LIN {X 0,Y 411.188,Z 252.265,A -85,B 0,C 180,E1 -10477.975,E2 -10477.975} C_VEL
LIN {X 0,Y 411.151,Z 252.273,A -85,B 0,C 180,E1 -10481.226,E2 -10481.226} C_VEL
LIN {X 0,Y 411.176,Z 252.271,A -85,B 0,C 180,E1 -10484.491,E2 -10484.491} C_VEL
LIN {X 0,Y 411.189,Z 252.269,A -85,B 0,C 180,E1 -10488.196,E2 -10488.196} C_VEL
LIN {X 0,Y 411.23,Z 252.345,A -85,B 0,C 180,E1 -10489.137,E2 -10489.137} C_VEL
LIN {X 0,Y 412.077,Z 257.26,A -85,B 0,C 180,E1 -10492.122,E2 -10492.122} C_VEL
LIN {X 0,Y 412.498,Z 261.588,A -85,B 0,C 180,E1 -10494.6,E2 -10494.6} C_VEL
LIN {X 0,Y 412.052,Z 268.088,A -85,B 0,C 180,E1 -10498.079,E2 -10498.079} C_VEL
LIN {X 0,Y 411.534,Z 274.615,A -85,B 0,C 180,E1 -10501.434,E2 -10501.434} C_VEL
LIN {X 0,Y 411.14,Z 281.666,A -85,B 0,C 180,E1 -10504.956,E2 -10504.956} C_VEL
LIN {X 0,Y 410.788,Z 288.71,A -85,B 0,C 180,E1 -10508.418,E2 -10508.418} C_VEL
LIN {X 0,Y 410.454,Z 296.177,A -85,B 0,C 180,E1 -10512.049,E2 -10512.049} C_VEL
LIN {X 0,Y 410.432,Z 296.997,A -85,B 0,C 180,E1 -10512.417,E2 -10512.417} C_VEL
LIN {X 0,Y 412.844,Z 310.073,A -85,B 0,C 180,E1 -10512.92,E2 -10512.92} C_VEL
LIN {X 0,Y 414.589,Z 322.997,A -85,B 0,C 180,E1 -10513.601,E2 -10513.601} C_VEL
LIN {X 0,Y 414.751,Z 328.091,A -85,B 0,C 180,E1 -10513.909,E2 -10513.909} C_VEL
LIN {X 0,Y 413.883,Z 340.094,A -85,B 0,C 180,E1 -10514.74,E2 -10514.74} C_VEL
LIN {X 0,Y 413.081,Z 351.078,A -85,B 0,C 180,E1 -10515.718,E2 -10515.718} C_VEL
LIN {X 0,Y 412.44,Z 360.002,A -85,B 0,C 180,E1 -10516.7,E2 -10516.7} C_VEL
LIN {X 0,Y 411.822,Z 369.176,A -85,B 0,C 180,E1 -10517.933,E2 -10517.933} C_VEL
LIN {X 0,Y 411.067,Z 378.113,A -85,B 0,C 180,E1 -10519.409,E2 -10519.409} C_VEL
LIN {X 0,Y 410.589,Z 385.309,A -85,B 0,C 180,E1 -10520.89,E2 -10520.89} C_VEL
LIN {X 0,Y 410.302,Z 390.167,A -85,B 0,C 180,E1 -10522.124,E2 -10522.124} C_VEL
LIN {X 0,Y 410.06,Z 395.319,A -85,B 0,C 180,E1 -10523.753,E2 -10523.753} C_VEL
LIN {X 0,Y 410.019,Z 398.5,A -85,B 0,C 180,E1 -10525.083,E2 -10525.083} C_VEL
LIN {X 0,Y 409.932,Z 400.361,A -85,B 0,C 180,E1 -10526.068,E2 -10526.068} C_VEL
LIN {X 0,Y 409.967,Z 402.755,A -85,B 0,C 180,E1 -10528.035,E2 -10528.035} C_VEL
LIN {X 0,Y 409.935,Z 403.362,A -85,B 0,C 180,E1 -10529.018,E2 -10529.018} C_VEL
LIN {X 0,Y 409.926,Z 403.578,A -85,B 0,C 180,E1 -10530,E2 -10530} C_VEL
LIN {X 0,Y 409.935,Z 403.36,A -85,B 0,C 180,E1 -10530.982,E2 -10530.982} C_VEL
LIN {X 0,Y 409.967,Z 402.753,A -85,B 0,C 180,E1 -10531.965,E2 -10531.965} C_VEL
LIN {X 0,Y 409.926,Z 401.755,A -85,B 0,C 180,E1 -10532.948,E2 -10532.948} C_VEL
LIN {X 0,Y 409.932,Z 400.356,A -85,B 0,C 180,E1 -10533.932,E2 -10533.932} C_VEL
LIN {X 0,Y 410.018,Z 397.418,A -85,B 0,C 180,E1 -10535.409,E2 -10535.409} C_VEL
LIN {X 0,Y 410.167,Z 393.441,A -85,B 0,C 180,E1 -10536.889,E2 -10536.889} C_VEL
LIN {X 0,Y 410.48,Z 387.326,A -85,B 0,C 180,E1 -10538.616,E2 -10538.616} C_VEL
LIN {X 0,Y 410.925,Z 380.646,A -85,B 0,C 180,E1 -10540.096,E2 -10540.096} C_VEL
LIN {X 0,Y 411.53,Z 372.36,A -85,B 0,C 180,E1 -10541.576,E2 -10541.576} C_VEL
LIN {X 0,Y 412.215,Z 363.868,A -85,B 0,C 180,E1 -10542.805,E2 -10542.805} C_VEL
LIN {X 0,Y 412.923,Z 353.392,A -85,B 0,C 180,E1 -10544.034,E2 -10544.034} C_VEL
LIN {X 0,Y 413.765,Z 341.563,A -85,B 0,C 180,E1 -10545.138,E2 -10545.138} C_VEL
LIN {X 0,Y 414.567,Z 329.887,A -85,B 0,C 180,E1 -10545.978,E2 -10545.978} C_VEL
LIN {X 0,Y 414.662,Z 323.977,A -85,B 0,C 180,E1 -10546.334,E2 -10546.334} C_VEL
LIN {X 0,Y 413.002,Z 311.075,A -85,B 0,C 180,E1 -10547.025,E2 -10547.025} C_VEL
LIN {X 0,Y 410.651,Z 298.45,A -85,B 0,C 180,E1 -10547.535,E2 -10547.535} C_VEL
LIN {X 0,Y 410.416,Z 296.925,A -85,B 0,C 180,E1 -10547.583,E2 -10547.583} C_VEL
LIN {X 0,Y 410.756,Z 289.772,A -85,B 0,C 180,E1 -10551.058,E2 -10551.058} C_VEL
LIN {X 0,Y 411.028,Z 283.293,A -85,B 0,C 180,E1 -10554.228,E2 -10554.228} C_VEL
LIN {X 0,Y 411.459,Z 275.668,A -85,B 0,C 180,E1 -10558.016,E2 -10558.016} C_VEL
LIN {X 0,Y 411.817,Z 270.22,A -85,B 0,C 180,E1 -10560.796,E2 -10560.796} C_VEL
LIN {X 0,Y 412.336,Z 263.709,A -85,B 0,C 180,E1 -10564.226,E2 -10564.226} C_VEL
LIN {X 0,Y 412.419,Z 260.479,A -85,B 0,C 180,E1 -10566.009,E2 -10566.009} C_VEL
LIN {X 0,Y 411.95,Z 256.526,A -85,B 0,C 180,E1 -10568.3,E2 -10568.3} C_VEL
LIN {X 0,Y 411.218,Z 252.27,A -85,B 0,C 180,E1 -10570.967,E2 -10570.967} C_VEL
LIN {X 0,Y 411.177,Z 252.269,A -85,B 0,C 180,E1 -10574.49,E2 -10574.49} C_VEL
LIN {X 0,Y 411.164,Z 252.268,A -85,B 0,C 180,E1 -10578.193,E2 -10578.193} C_VEL
LIN {X 0,Y 411.195,Z 252.262,A -85,B 0,C 180,E1 -10581.833,E2 -10581.833} C_VEL
LIN {X 0,Y 411.212,Z 252.262,A -85,B 0,C 180,E1 -10585.122,E2 -10585.122} C_VEL
LIN {X 0,Y 411.167,Z 252.27,A -85,B 0,C 180,E1 -10588.003,E2 -10588.003} C_VEL
LIN {X 0,Y 411.194,Z 252.263,A -85,B 0,C 180,E1 -10591.408,E2 -10591.408} C_VEL
LIN {X 0,Y 411.213,Z 252.26,A -85,B 0,C 180,E1 -10594.934,E2 -10594.934} C_VEL
LIN {X 0,Y 411.205,Z 252.267,A -85,B 0,C 180,E1 -10597.913,E2 -10597.913} C_VEL
LIN {X 0,Y 411.226,Z 252.259,A -85,B 0,C 180,E1 -10601.052,E2 -10601.052} C_VEL
LIN {X 0,Y 411.256,Z 252.258,A -85,B 0,C 180,E1 -10604.132,E2 -10604.132} C_VEL
LIN {X 0,Y 411.305,Z 252.251,A -85,B 0,C 180,E1 -10607.166,E2 -10607.166} C_VEL
LIN {X 0,Y 411.29,Z 252.251,A -85,B 0,C 180,E1 -10610.161,E2 -10610.161} C_VEL
LIN {X 0,Y 411.438,Z 252.235,A -85,B 0,C 180,E1 -10613.133,E2 -10613.133} C_VEL
LIN {X 0,Y 411.31,Z 252.252,A -85,B 0,C 180,E1 -10615.099,E2 -10615.099} C_VEL
LIN {X 0,Y 411.513,Z 252.224,A -85,B 0,C 180,E1 -10618.043,E2 -10618.043} C_VEL
LIN {X 0,Y 411.637,Z 252.208,A -85,B 0,C 180,E1 -10620,E2 -10620} C_VEL
LIN {X 0,Y 411.438,Z 252.236,A -85,B 0,C 180,E1 -10622.937,E2 -10622.937} C_VEL
LIN {X 0,Y 411.435,Z 252.237,A -85,B 0,C 180,E1 -10626.867,E2 -10626.867} C_VEL
LIN {X 0,Y 411.294,Z 252.25,A -85,B 0,C 180,E1 -10629.839,E2 -10629.839} C_VEL
LIN {X 0,Y 411.307,Z 252.253,A -85,B 0,C 180,E1 -10633.104,E2 -10633.104} C_VEL
LIN {X 0,Y 411.259,Z 252.259,A -85,B 0,C 180,E1 -10636.889,E2 -10636.889} C_VEL
LIN {X 0,Y 411.232,Z 252.259,A -85,B 0,C 180,E1 -10639.987,E2 -10639.987} C_VEL
LIN {X 0,Y 411.198,Z 252.263,A -85,B 0,C 180,E1 -10643.148,E2 -10643.148} C_VEL
LIN {X 0,Y 411.238,Z 252.261,A -85,B 0,C 180,E1 -10646.381,E2 -10646.381} C_VEL
LIN {X 0,Y 411.202,Z 252.264,A -85,B 0,C 180,E1 -10649.713,E2 -10649.713} C_VEL
LIN {X 0,Y 411.205,Z 252.261,A -85,B 0,C 180,E1 -10653.156,E2 -10653.156} C_VEL
LIN {X 0,Y 411.193,Z 252.264,A -85,B 0,C 180,E1 -10656.552,E2 -10656.552} C_VEL
LIN {X 0,Y 411.208,Z 252.266,A -85,B 0,C 180,E1 -10659.727,E2 -10659.727} C_VEL
LIN {X 0,Y 411.172,Z 252.267,A -85,B 0,C 180,E1 -10663.134,E2 -10663.134} C_VEL
LIN {X 0,Y 411.163,Z 252.271,A -85,B 0,C 180,E1 -10665.882,E2 -10665.882} C_VEL
LIN {X 0,Y 411.159,Z 252.272,A -85,B 0,C 180,E1 -10669.493,E2 -10669.493} C_VEL
LIN {X 0,Y 411.185,Z 252.265,A -85,B 0,C 180,E1 -10672.025,E2 -10672.025} C_VEL
LIN {X 0,Y 411.079,Z 252.531,A -85,B 0,C 180,E1 -10674.459,E2 -10674.459} C_VEL
LIN {X 0,Y 411.063,Z 255.493,A -85,B 0,C 180,E1 -10676.905,E2 -10676.905} C_VEL
LIN {X 0,Y 410.848,Z 259.693,A -85,B 0,C 180,E1 -10680.259,E2 -10680.259} C_VEL
LIN {X 0,Y 410.661,Z 263.957,A -85,B 0,C 180,E1 -10683.579,E2 -10683.579} C_VEL
LIN {X 0,Y 410.513,Z 268.258,A -85,B 0,C 180,E1 -10686.811,E2 -10686.811} C_VEL
LIN {X 0,Y 410.384,Z 273.156,A -85,B 0,C 180,E1 -10690.373,E2 -10690.373} C_VEL
LIN {X 0,Y 410.298,Z 276.157,A -85,B 0,C 180,E1 -10692.466,E2 -10692.466} C_VEL
LIN {X 0,Y 413.974,Z 291.968,A -85,B 0,C 180,E1 -10693.193,E2 -10693.193} C_VEL
LIN {X 0,Y 415.297,Z 299.636,A -85,B 0,C 180,E1 -10693.629,E2 -10693.629} C_VEL
LIN {X 0,Y 414.754,Z 312.054,A -85,B 0,C 180,E1 -10694.395,E2 -10694.395} C_VEL
LIN {X 0,Y 414.084,Z 322.819,A -85,B 0,C 180,E1 -10695.251,E2 -10695.251} C_VEL
LIN {X 0,Y 413.333,Z 333.788,A -85,B 0,C 180,E1 -10696.354,E2 -10696.354} C_VEL
LIN {X 0,Y 412.607,Z 342.694,A -85,B 0,C 180,E1 -10697.457,E2 -10697.457} C_VEL
LIN {X 0,Y 412.017,Z 350.86,A -85,B 0,C 180,E1 -10698.687,E2 -10698.687} C_VEL
LIN {X 0,Y 411.344,Z 358.861,A -85,B 0,C 180,E1 -10700.163,E2 -10700.163} C_VEL
LIN {X 0,Y 410.816,Z 365.285,A -85,B 0,C 180,E1 -10701.639,E2 -10701.639} C_VEL
LIN {X 0,Y 410.435,Z 370.888,A -85,B 0,C 180,E1 -10703.293,E2 -10703.293} C_VEL
LIN {X 0,Y 410.168,Z 375.396,A -85,B 0,C 180,E1 -10705.085,E2 -10705.085} C_VEL
LIN {X 0,Y 410.048,Z 377.257,A -85,B 0,C 180,E1 -10706.069,E2 -10706.069} C_VEL
LIN {X 0,Y 410.056,Z 378.656,A -85,B 0,C 180,E1 -10707.053,E2 -10707.053} C_VEL
LIN {X 0,Y 410.012,Z 379.652,A -85,B 0,C 180,E1 -10708.035,E2 -10708.035} C_VEL
LIN {X 0,Y 409.927,Z 380.501,A -85,B 0,C 180,E1 -10710,E2 -10710} C_VEL
LIN {X 0,Y 409.939,Z 380.313,A -85,B 0,C 180,E1 -10710.982,E2 -10710.982} C_VEL
LIN {X 0,Y 410.012,Z 379.727,A -85,B 0,C 180,E1 -10711.965,E2 -10711.965} C_VEL
LIN {X 0,Y 410.055,Z 378.761,A -85,B 0,C 180,E1 -10712.947,E2 -10712.947} C_VEL
LIN {X 0,Y 410.044,Z 377.408,A -85,B 0,C 180,E1 -10713.931,E2 -10713.931} C_VEL
LIN {X 0,Y 410.271,Z 374.541,A -85,B 0,C 180,E1 -10715.406,E2 -10715.406} C_VEL
LIN {X 0,Y 410.501,Z 370.656,A -85,B 0,C 180,E1 -10716.883,E2 -10716.883} C_VEL
LIN {X 0,Y 410.771,Z 365.645,A -85,B 0,C 180,E1 -10718.362,E2 -10718.362} C_VEL
LIN {X 0,Y 410.979,Z 362.945,A -85,B 0,C 180,E1 -10719.033,E2 -10719.033} C_VEL
LIN {X 0,Y 410.576,Z 359.967,A -85,B 0,C 180,E1 -10719.744,E2 -10719.744} C_VEL
LIN {X 0,Y 408.212,Z 354.758,A -85,B 0,C 180,E1 -10720.88,E2 -10720.88} C_VEL
LIN {X 0,Y 405.881,Z 348.9,A -85,B 0,C 180,E1 -10721.96,E2 -10721.96} C_VEL
LIN {X 0,Y 405.53,Z 344.902,A -85,B 0,C 180,E1 -10722.575,E2 -10722.575} C_VEL
LIN {X 0,Y 406.413,Z 334.803,A -85,B 0,C 180,E1 -10723.883,E2 -10723.883} C_VEL
LIN {X 0,Y 407.126,Z 324.064,A -85,B 0,C 180,E1 -10725.007,E2 -10725.007} C_VEL
LIN {X 0,Y 407.865,Z 313.593,A -85,B 0,C 180,E1 -10725.875,E2 -10725.875} C_VEL
LIN {X 0,Y 408.551,Z 301.428,A -85,B 0,C 180,E1 -10726.657,E2 -10726.657} C_VEL
LIN {X 0,Y 406.421,Z 289.764,A -85,B 0,C 180,E1 -10727.331,E2 -10727.331} C_VEL
LIN {X 0,Y 403.215,Z 276.357,A -85,B 0,C 180,E1 -10727.947,E2 -10727.947} C_VEL
LIN {X 0,Y 403.316,Z 272.909,A -85,B 0,C 180,E1 -10730.396,E2 -10730.396} C_VEL
LIN {X 0,Y 403.459,Z 268.567,A -85,B 0,C 180,E1 -10733.619,E2 -10733.619} C_VEL
LIN {X 0,Y 403.666,Z 264.253,A -85,B 0,C 180,E1 -10736.915,E2 -10736.915} C_VEL
LIN {X 0,Y 403.828,Z 259.977,A -85,B 0,C 180,E1 -10740.312,E2 -10740.312} C_VEL
LIN {X 0,Y 403.984,Z 255.665,A -85,B 0,C 180,E1 -10743.828,E2 -10743.828} C_VEL
LIN {X 0,Y 404.041,Z 254.063,A -85,B 0,C 180,E1 -10745.161,E2 -10745.161} C_VEL
LIN {X 0,Y 404.055,Z 253.156,A -85,B 0,C 180,E1 -10746.256,E2 -10746.256} C_VEL
LIN {X 0,Y 404.136,Z 253.146,A -85,B 0,C 180,E1 -10748.759,E2 -10748.759} C_VEL
LIN {X 0,Y 404.108,Z 253.145,A -85,B 0,C 180,E1 -10751.597,E2 -10751.597} C_VEL
LIN {X 0,Y 404.145,Z 253.145,A -85,B 0,C 180,E1 -10754.522,E2 -10754.522} C_VEL
LIN {X 0,Y 404.135,Z 253.142,A -85,B 0,C 180,E1 -10757.295,E2 -10757.295} C_VEL
LIN {X 0,Y 404.172,Z 253.141,A -85,B 0,C 180,E1 -10759.955,E2 -10759.955} C_VEL
LIN {X 0,Y 404.138,Z 253.141,A -85,B 0,C 180,E1 -10763.125,E2 -10763.125} C_VEL
LIN {X 0,Y 404.147,Z 253.144,A -85,B 0,C 180,E1 -10766.188,E2 -10766.188} C_VEL
LIN {X 0,Y 404.148,Z 253.145,A -85,B 0,C 180,E1 -10769.715,E2 -10769.715} C_VEL
LIN {X 0,Y 404.198,Z 253.135,A -85,B 0,C 180,E1 -10773.123,E2 -10773.123} C_VEL
LIN {X 0,Y 404.177,Z 253.14,A -85,B 0,C 180,E1 -10775.334,E2 -10775.334} C_VEL
LIN {X 0,Y 404.141,Z 253.14,A -85,B 0,C 180,E1 -10778.581,E2 -10778.581} C_VEL
LIN {X 0,Y 404.206,Z 253.136,A -85,B 0,C 180,E1 -10781.762,E2 -10781.762} C_VEL
LIN {X 0,Y 404.205,Z 253.135,A -85,B 0,C 180,E1 -10784.882,E2 -10784.882} C_VEL
LIN {X 0,Y 404.26,Z 253.127,A -85,B 0,C 180,E1 -10787.959,E2 -10787.959} C_VEL
LIN {X 0,Y 404.27,Z 253.129,A -85,B 0,C 180,E1 -10790.998,E2 -10790.998} C_VEL
LIN {X 0,Y 404.398,Z 253.108,A -85,B 0,C 180,E1 -10794.015,E2 -10794.015} C_VEL
LIN {X 0,Y 404.477,Z 253.099,A -85,B 0,C 180,E1 -10798.008,E2 -10798.008} C_VEL
LIN {X 0,Y 404.413,Z 253.111,A -85,B 0,C 180,E1 -10800.996,E2 -10800.996} C_VEL
LIN {X 0,Y 404.419,Z 253.111,A -85,B 0,C 180,E1 -10802.988,E2 -10802.988} C_VEL
LIN {X 0,Y 404.417,Z 253.108,A -85,B 0,C 180,E1 -10805.985,E2 -10805.985} C_VEL
LIN {X 0,Y 404.262,Z 253.127,A -85,B 0,C 180,E1 -10809.002,E2 -10809.002} C_VEL
LIN {X 0,Y 404.251,Z 253.13,A -85,B 0,C 180,E1 -10812.042,E2 -10812.042} C_VEL
LIN {X 0,Y 404.208,Z 253.133,A -85,B 0,C 180,E1 -10815.118,E2 -10815.118} C_VEL
LIN {X 0,Y 404.213,Z 253.137,A -85,B 0,C 180,E1 -10818.238,E2 -10818.238} C_VEL
LIN {X 0,Y 404.141,Z 253.142,A -85,B 0,C 180,E1 -10821.419,E2 -10821.419} C_VEL
LIN {X 0,Y 404.151,Z 253.14,A -85,B 0,C 180,E1 -10824.667,E2 -10824.667} C_VEL
LIN {X 0,Y 404.131,Z 253.146,A -85,B 0,C 180,E1 -10828.005,E2 -10828.005} C_VEL
LIN {X 0,Y 404.146,Z 253.142,A -85,B 0,C 180,E1 -10830.285,E2 -10830.285} C_VEL
LIN {X 0,Y 404.147,Z 253.145,A -85,B 0,C 180,E1 -10833.812,E2 -10833.812} C_VEL
LIN {X 0,Y 404.136,Z 253.142,A -85,B 0,C 180,E1 -10836.874,E2 -10836.874} C_VEL
LIN {X 0,Y 404.118,Z 253.144,A -85,B 0,C 180,E1 -10840.075,E2 -10840.075} C_VEL
LIN {X 0,Y 404.146,Z 253.145,A -85,B 0,C 180,E1 -10843.082,E2 -10843.082} C_VEL
LIN {X 0,Y 404.15,Z 253.145,A -85,B 0,C 180,E1 -10845.926,E2 -10845.926} C_VEL
LIN {X 0,Y 404.203,Z 253.254,A -85,B 0,C 180,E1 -10848.889,E2 -10848.889} C_VEL
LIN {X 0,Y 405.051,Z 258.256,A -85,B 0,C 180,E1 -10851.995,E2 -10851.995} C_VEL
LIN {X 0,Y 405.482,Z 262.634,A -85,B 0,C 180,E1 -10854.551,E2 -10854.551} C_VEL
LIN {X 0,Y 405.056,Z 267.954,A -85,B 0,C 180,E1 -10857.461,E2 -10857.461} C_VEL
LIN {X 0,Y 404.543,Z 274.461,A -85,B 0,C 180,E1 -10860.893,E2 -10860.893} C_VEL
LIN {X 0,Y 404.13,Z 280.994,A -85,B 0,C 180,E1 -10864.23,E2 -10864.23} C_VEL
LIN {X 0,Y 403.815,Z 287.456,A -85,B 0,C 180,E1 -10867.487,E2 -10867.487} C_VEL
LIN {X 0,Y 403.464,Z 293.871,A -85,B 0,C 180,E1 -10870.673,E2 -10870.673} C_VEL
LIN {X 0,Y 403.374,Z 296.889,A -85,B 0,C 180,E1 -10872.1,E2 -10872.1} C_VEL
LIN {X 0,Y 405.849,Z 309.951,A -85,B 0,C 180,E1 -10872.619,E2 -10872.619} C_VEL
LIN {X 0,Y 407.574,Z 322.49,A -85,B 0,C 180,E1 -10873.293,E2 -10873.293} C_VEL
LIN {X 0,Y 407.896,Z 328.234,A -85,B 0,C 180,E1 -10873.653,E2 -10873.653} C_VEL
LIN {X 0,Y 407.006,Z 339.897,A -85,B 0,C 180,E1 -10874.476,E2 -10874.476} C_VEL
LIN {X 0,Y 406.142,Z 351.347,A -85,B 0,C 180,E1 -10875.52,E2 -10875.52} C_VEL
LIN {X 0,Y 405.401,Z 361.819,A -85,B 0,C 180,E1 -10876.728,E2 -10876.728} C_VEL
LIN {X 0,Y 404.697,Z 370.61,A -85,B 0,C 180,E1 -10877.972,E2 -10877.972} C_VEL
LIN {X 0,Y 403.975,Z 379.236,A -85,B 0,C 180,E1 -10879.475,E2 -10879.475} C_VEL
LIN {X 0,Y 403.495,Z 386.135,A -85,B 0,C 180,E1 -10880.981,E2 -10880.981} C_VEL
LIN {X 0,Y 403.148,Z 391.664,A -85,B 0,C 180,E1 -10882.487,E2 -10882.487} C_VEL
LIN {X 0,Y 402.943,Z 396.002,A -85,B 0,C 180,E1 -10883.993,E2 -10883.993} C_VEL
LIN {X 0,Y 402.932,Z 398.301,A -85,B 0,C 180,E1 -10884.997,E2 -10884.997} C_VEL
LIN {X 0,Y 402.852,Z 400.161,A -85,B 0,C 180,E1 -10885.998,E2 -10885.998} C_VEL
LIN {X 0,Y 402.865,Z 402.555,A -85,B 0,C 180,E1 -10888,E2 -10888} C_VEL
LIN {X 0,Y 402.862,Z 403.163,A -85,B 0,C 180,E1 -10889,E2 -10889} C_VEL
LIN {X 0,Y 402.851,Z 403.378,A -85,B 0,C 180,E1 -10890,E2 -10890} C_VEL
LIN {X 0,Y 402.862,Z 403.161,A -85,B 0,C 180,E1 -10890.999,E2 -10890.999} C_VEL
LIN {X 0,Y 402.865,Z 402.552,A -85,B 0,C 180,E1 -10891.999,E2 -10891.999} C_VEL
LIN {X 0,Y 402.852,Z 400.156,A -85,B 0,C 180,E1 -10894.001,E2 -10894.001} C_VEL
LIN {X 0,Y 402.916,Z 397.216,A -85,B 0,C 180,E1 -10895.505,E2 -10895.505} C_VEL
LIN {X 0,Y 403.08,Z 393.239,A -85,B 0,C 180,E1 -10897.01,E2 -10897.01} C_VEL
LIN {X 0,Y 403.419,Z 387.123,A -85,B 0,C 180,E1 -10898.768,E2 -10898.768} C_VEL
LIN {X 0,Y 403.916,Z 380.444,A -85,B 0,C 180,E1 -10900.273,E2 -10900.273} C_VEL
LIN {X 0,Y 404.553,Z 372.157,A -85,B 0,C 180,E1 -10901.778,E2 -10901.778} C_VEL
LIN {X 0,Y 405.257,Z 363.665,A -85,B 0,C 180,E1 -10903.029,E2 -10903.029} C_VEL
LIN {X 0,Y 405.98,Z 353.406,A -85,B 0,C 180,E1 -10904.256,E2 -10904.256} C_VEL
LIN {X 0,Y 406.795,Z 342.788,A -85,B 0,C 180,E1 -10905.276,E2 -10905.276} C_VEL
LIN {X 0,Y 407.64,Z 331.601,A -85,B 0,C 180,E1 -10906.127,E2 -10906.127} C_VEL
LIN {X 0,Y 407.933,Z 326.356,A -85,B 0,C 180,E1 -10906.459,E2 -10906.459} C_VEL
LIN {X 0,Y 406.395,Z 313.694,A -85,B 0,C 180,E1 -10907.19,E2 -10907.19} C_VEL
LIN {X 0,Y 404.141,Z 300.805,A -85,B 0,C 180,E1 -10907.754,E2 -10907.754} C_VEL
LIN {X 0,Y 403.377,Z 296.701,A -85,B 0,C 180,E1 -10907.916,E2 -10907.916} C_VEL
LIN {X 0,Y 403.7,Z 289.587,A -85,B 0,C 180,E1 -10911.444,E2 -10911.444} C_VEL
LIN {X 0,Y 404.01,Z 283.126,A -85,B 0,C 180,E1 -10914.676,E2 -10914.676} C_VEL
LIN {X 0,Y 404.396,Z 276.599,A -85,B 0,C 180,E1 -10917.984,E2 -10917.984} C_VEL
LIN {X 0,Y 404.785,Z 271.16,A -85,B 0,C 180,E1 -10920.81,E2 -10920.81} C_VEL
LIN {X 0,Y 405.347,Z 264.678,A -85,B 0,C 180,E1 -10924.298,E2 -10924.298} C_VEL
LIN {X 0,Y 405.406,Z 261.442,A -85,B 0,C 180,E1 -10926.115,E2 -10926.115} C_VEL
LIN {X 0,Y 404.853,Z 257.144,A -85,B 0,C 180,E1 -10928.678,E2 -10928.678} C_VEL
LIN {X 0,Y 404.153,Z 253.148,A -85,B 0,C 180,E1 -10931.198,E2 -10931.198} C_VEL
LIN {X 0,Y 404.146,Z 253.144,A -85,B 0,C 180,E1 -10934.522,E2 -10934.522} C_VEL
LIN {X 0,Y 404.125,Z 253.144,A -85,B 0,C 180,E1 -10937.294,E2 -10937.294} C_VEL
LIN {X 0,Y 404.133,Z 253.142,A -85,B 0,C 180,E1 -10939.951,E2 -10939.951} C_VEL
LIN {X 0,Y 404.135,Z 253.143,A -85,B 0,C 180,E1 -10943.125,E2 -10943.125} C_VEL
LIN {X 0,Y 404.146,Z 253.145,A -85,B 0,C 180,E1 -10946.188,E2 -10946.188} C_VEL
LIN {X 0,Y 404.145,Z 253.142,A -85,B 0,C 180,E1 -10949.715,E2 -10949.715} C_VEL
LIN {X 0,Y 404.13,Z 253.142,A -85,B 0,C 180,E1 -10953.118,E2 -10953.118} C_VEL
LIN {X 0,Y 404.151,Z 253.142,A -85,B 0,C 180,E1 -10956.424,E2 -10956.424} C_VEL
LIN {X 0,Y 404.193,Z 253.139,A -85,B 0,C 180,E1 -10959.874,E2 -10959.874} C_VEL
LIN {X 0,Y 404.217,Z 253.132,A -85,B 0,C 180,E1 -10962.993,E2 -10962.993} C_VEL
LIN {X 0,Y 404.284,Z 253.124,A -85,B 0,C 180,E1 -10966.939,E2 -10966.939} C_VEL
LIN {X 0,Y 404.256,Z 253.128,A -85,B 0,C 180,E1 -10969.988,E2 -10969.988} C_VEL
LIN {X 0,Y 404.387,Z 253.112,A -85,B 0,C 180,E1 -10973.012,E2 -10973.012} C_VEL
LIN {X 0,Y 404.281,Z 253.126,A -85,B 0,C 180,E1 -10975.014,E2 -10975.014} C_VEL
LIN {X 0,Y 404.482,Z 253.1,A -85,B 0,C 180,E1 -10978.009,E2 -10978.009} C_VEL
LIN {X 0,Y 404.607,Z 253.084,A -85,B 0,C 180,E1 -10980,E2 -10980} C_VEL
LIN {X 0,Y 404.397,Z 253.113,A -85,B 0,C 180,E1 -10982.989,E2 -10982.989} C_VEL
LIN {X 0,Y 404.385,Z 253.116,A -85,B 0,C 180,E1 -10986.988,E2 -10986.988} C_VEL
LIN {X 0,Y 404.255,Z 253.131,A -85,B 0,C 180,E1 -10991.025,E2 -10991.025} C_VEL
LIN {X 0,Y 404.212,Z 253.133,A -85,B 0,C 180,E1 -10994.088,E2 -10994.088} C_VEL
LIN {X 0,Y 404.204,Z 253.135,A -85,B 0,C 180,E1 -10997.193,E2 -10997.193} C_VEL
LIN {X 0,Y 404.165,Z 253.142,A -85,B 0,C 180,E1 -11000.352,E2 -11000.352} C_VEL
LIN {X 0,Y 404.165,Z 253.138,A -85,B 0,C 180,E1 -11003.575,E2 -11003.575} C_VEL
LIN {X 0,Y 404.185,Z 253.137,A -85,B 0,C 180,E1 -11005.767,E2 -11005.767} C_VEL
LIN {X 0,Y 404.197,Z 253.138,A -85,B 0,C 180,E1 -11008,E2 -11008} C_VEL
LIN {X 0,Y 404.14,Z 253.143,A -85,B 0,C 180,E1 -11011.558,E2 -11011.558} C_VEL
LIN {X 0,Y 404.175,Z 253.136,A -85,B 0,C 180,E1 -11015.017,E2 -11015.017} C_VEL
LIN {X 0,Y 404.15,Z 253.14,A -85,B 0,C 180,E1 -11018.758,E2 -11018.758} C_VEL
LIN {X 0,Y 404.12,Z 253.148,A -85,B 0,C 180,E1 -11021.599,E2 -11021.599} C_VEL
LIN {X 0,Y 404.145,Z 253.141,A -85,B 0,C 180,E1 -11024.522,E2 -11024.522} C_VEL
LIN {X 0,Y 404.121,Z 253.147,A -85,B 0,C 180,E1 -11027.293,E2 -11027.293} C_VEL
LIN {X 0,Y 404.133,Z 253.144,A -85,B 0,C 180,E1 -11029.951,E2 -11029.951} C_VEL
LIN {X 0,Y 404.108,Z 253.151,A -85,B 0,C 180,E1 -11033.131,E2 -11033.131} C_VEL
LIN {X 0,Y 404.083,Z 253.153,A -85,B 0,C 180,E1 -11033.748,E2 -11033.748} C_VEL
LIN {X 0,Y 404.072,Z 254.088,A -85,B 0,C 180,E1 -11034.973,E2 -11034.973} C_VEL
LIN {X 0,Y 403.98,Z 256.962,A -85,B 0,C 180,E1 -11037.364,E2 -11037.364} C_VEL
LIN {X 0,Y 403.766,Z 261.256,A -85,B 0,C 180,E1 -11040.832,E2 -11040.832} C_VEL
LIN {X 0,Y 403.564,Z 265.535,A -85,B 0,C 180,E1 -11044.191,E2 -11044.191} C_VEL
LIN {X 0,Y 403.42,Z 269.87,A -85,B 0,C 180,E1 -11047.464,E2 -11047.464} C_VEL
LIN {X 0,Y 403.295,Z 274.252,A -85,B 0,C 180,E1 -11050.664,E2 -11050.664} C_VEL
LIN {X 0,Y 403.236,Z 276.383,A -85,B 0,C 180,E1 -11052.171,E2 -11052.171} C_VEL
LIN {X 0,Y 406.356,Z 289.43,A -85,B 0,C 180,E1 -11052.75,E2 -11052.75} C_VEL
LIN {X 0,Y 408.45,Z 300.6,A -85,B 0,C 180,E1 -11053.39,E2 -11053.39} C_VEL
LIN {X 0,Y 407.92,Z 312.261,A -85,B 0,C 180,E1 -11054.127,E2 -11054.127} C_VEL
LIN {X 0,Y 407.225,Z 323.024,A -85,B 0,C 180,E1 -11054.997,E2 -11054.997} C_VEL
LIN {X 0,Y 406.435,Z 333.992,A -85,B 0,C 180,E1 -11056.118,E2 -11056.118} C_VEL
LIN {X 0,Y 405.558,Z 344.67,A -85,B 0,C 180,E1 -11057.49,E2 -11057.49} C_VEL
LIN {X 0,Y 404.921,Z 352.541,A -85,B 0,C 180,E1 -11058.74,E2 -11058.74} C_VEL
LIN {X 0,Y 404.236,Z 360.236,A -85,B 0,C 180,E1 -11060.241,E2 -11060.241} C_VEL
LIN {X 0,Y 403.635,Z 367.296,A -85,B 0,C 180,E1 -11061.993,E2 -11061.993} C_VEL
LIN {X 0,Y 403.347,Z 371.464,A -85,B 0,C 180,E1 -11063.307,E2 -11063.307} C_VEL
LIN {X 0,Y 403.113,Z 375.596,A -85,B 0,C 180,E1 -11064.999,E2 -11064.999} C_VEL
LIN {X 0,Y 402.966,Z 377.458,A -85,B 0,C 180,E1 -11066,E2 -11066} C_VEL
LIN {X 0,Y 402.959,Z 378.856,A -85,B 0,C 180,E1 -11067.001,E2 -11067.001} C_VEL
LIN {X 0,Y 402.944,Z 379.851,A -85,B 0,C 180,E1 -11068.001,E2 -11068.001} C_VEL
LIN {X 0,Y 402.852,Z 380.7,A -85,B 0,C 180,E1 -11070,E2 -11070} C_VEL
LIN {X 0,Y 402.867,Z 380.512,A -85,B 0,C 180,E1 -11071,E2 -11071} C_VEL
LIN {X 0,Y 402.944,Z 379.926,A -85,B 0,C 180,E1 -11071.999,E2 -11071.999} C_VEL
LIN {X 0,Y 402.958,Z 378.961,A -85,B 0,C 180,E1 -11072.999,E2 -11072.999} C_VEL
LIN {X 0,Y 402.962,Z 377.607,A -85,B 0,C 180,E1 -11074.001,E2 -11074.001} C_VEL
LIN {X 0,Y 403.199,Z 374.74,A -85,B 0,C 180,E1 -11075.501,E2 -11075.501} C_VEL
LIN {X 0,Y 403.452,Z 370.854,A -85,B 0,C 180,E1 -11077.004,E2 -11077.004} C_VEL
LIN {X 0,Y 403.729,Z 365.844,A -85,B 0,C 180,E1 -11078.509,E2 -11078.509} C_VEL
LIN {X 0,Y 404.289,Z 359.531,A -85,B 0,C 180,E1 -11080.011,E2 -11080.011} C_VEL
LIN {X 0,Y 404.969,Z 351.628,A -85,B 0,C 180,E1 -11081.512,E2 -11081.512} C_VEL
LIN {X 0,Y 405.53,Z 344.902,A -85,B 0,C 180,E1 -11082.575,E2 -11082.575} C_VEL
LIN {X 0,Y 405.199,Z 340.794,A -85,B 0,C 180,E1 -11083.169,E2 -11083.169} C_VEL
LIN {X 0,Y 401.949,Z 331.02,A -85,B 0,C 180,E1 -11084.497,E2 -11084.497} C_VEL
LIN {X 0,Y 400.524,Z 324.93,A -85,B 0,C 180,E1 -11085.192,E2 -11085.192} C_VEL
LIN {X 0,Y 400.436,Z 321.651,A -85,B 0,C 180,E1 -11085.507,E2 -11085.507} C_VEL
LIN {X 0,Y 401.258,Z 310.555,A -85,B 0,C 180,E1 -11086.384,E2 -11086.384} C_VEL
LIN {X 0,Y 401.722,Z 302.266,A -85,B 0,C 180,E1 -11086.911,E2 -11086.911} C_VEL
LIN {X 0,Y 399.473,Z 290.353,A -85,B 0,C 180,E1 -11087.625,E2 -11087.625} C_VEL
LIN {X 0,Y 396.28,Z 277.374,A -85,B 0,C 180,E1 -11088.231,E2 -11088.231} C_VEL
LIN {X 0,Y 396.156,Z 276.539,A -85,B 0,C 180,E1 -11088.287,E2 -11088.287} C_VEL
LIN {X 0,Y 396.25,Z 273.094,A -85,B 0,C 180,E1 -11090.777,E2 -11090.777} C_VEL
LIN {X 0,Y 396.436,Z 268.742,A -85,B 0,C 180,E1 -11094.063,E2 -11094.063} C_VEL
LIN {X 0,Y 396.634,Z 264.164,A -85,B 0,C 180,E1 -11097.63,E2 -11097.63} C_VEL
LIN {X 0,Y 396.808,Z 260.131,A -85,B 0,C 180,E1 -11100.906,E2 -11100.906} C_VEL
LIN {X 0,Y 396.967,Z 255.777,A -85,B 0,C 180,E1 -11104.509,E2 -11104.509} C_VEL
LIN {X 0,Y 396.997,Z 254.347,A -85,B 0,C 180,E1 -11105.746,E2 -11105.746} C_VEL
LIN {X 0,Y 397.073,Z 254.025,A -85,B 0,C 180,E1 -11107.204,E2 -11107.204} C_VEL
LIN {X 0,Y 397.056,Z 254.028,A -85,B 0,C 180,E1 -11110.437,E2 -11110.437} C_VEL
LIN {X 0,Y 397.089,Z 254.02,A -85,B 0,C 180,E1 -11113.65,E2 -11113.65} C_VEL
LIN {X 0,Y 397.103,Z 254.022,A -85,B 0,C 180,E1 -11116.521,E2 -11116.521} C_VEL
LIN {X 0,Y 397.115,Z 254.02,A -85,B 0,C 180,E1 -11120.423,E2 -11120.423} C_VEL
LIN {X 0,Y 397.11,Z 254.02,A -85,B 0,C 180,E1 -11124.265,E2 -11124.265} C_VEL
LIN {X 0,Y 397.117,Z 254.016,A -85,B 0,C 180,E1 -11126.727,E2 -11126.727} C_VEL
LIN {X 0,Y 397.127,Z 254.017,A -85,B 0,C 180,E1 -11130.296,E2 -11130.296} C_VEL
LIN {X 0,Y 397.197,Z 254.006,A -85,B 0,C 180,E1 -11132.61,E2 -11132.61} C_VEL
LIN {X 0,Y 397.131,Z 254.017,A -85,B 0,C 180,E1 -11135.982,E2 -11135.982} C_VEL
LIN {X 0,Y 397.142,Z 254.016,A -85,B 0,C 180,E1 -11139.705,E2 -11139.705} C_VEL
LIN {X 0,Y 397.185,Z 254.009,A -85,B 0,C 180,E1 -11142.845,E2 -11142.845} C_VEL
LIN {X 0,Y 397.232,Z 254.003,A -85,B 0,C 180,E1 -11146.703,E2 -11146.703} C_VEL
LIN {X 0,Y 397.221,Z 254.004,A -85,B 0,C 180,E1 -11149.809,E2 -11149.809} C_VEL
LIN {X 0,Y 397.334,Z 253.993,A -85,B 0,C 180,E1 -11152.888,E2 -11152.888} C_VEL
LIN {X 0,Y 397.243,Z 254.005,A -85,B 0,C 180,E1 -11154.925,E2 -11154.925} C_VEL
LIN {X 0,Y 397.445,Z 253.975,A -85,B 0,C 180,E1 -11157.973,E2 -11157.973} C_VEL
LIN {X 0,Y 397.378,Z 253.988,A -85,B 0,C 180,E1 -11161.013,E2 -11161.013} C_VEL
LIN {X 0,Y 397.378,Z 253.987,A -85,B 0,C 180,E1 -11163.041,E2 -11163.041} C_VEL
LIN {X 0,Y 397.367,Z 253.987,A -85,B 0,C 180,E1 -11166.092,E2 -11166.092} C_VEL
LIN {X 0,Y 397.232,Z 254.001,A -85,B 0,C 180,E1 -11169.162,E2 -11169.162} C_VEL
LIN {X 0,Y 397.216,Z 254.009,A -85,B 0,C 180,E1 -11172.258,E2 -11172.258} C_VEL
LIN {X 0,Y 397.182,Z 254.008,A -85,B 0,C 180,E1 -11175.392,E2 -11175.392} C_VEL
LIN {X 0,Y 397.165,Z 254.012,A -85,B 0,C 180,E1 -11178.573,E2 -11178.573} C_VEL
LIN {X 0,Y 397.098,Z 254.022,A -85,B 0,C 180,E1 -11181.818,E2 -11181.818} C_VEL
LIN {X 0,Y 397.099,Z 254.018,A -85,B 0,C 180,E1 -11185.136,E2 -11185.136} C_VEL
LIN {X 0,Y 397.08,Z 254.021,A -85,B 0,C 180,E1 -11188.547,E2 -11188.547} C_VEL
LIN {X 0,Y 397.084,Z 254.025,A -85,B 0,C 180,E1 -11191.836,E2 -11191.836} C_VEL
LIN {X 0,Y 397.127,Z 254.015,A -85,B 0,C 180,E1 -11194.493,E2 -11194.493} C_VEL
LIN {X 0,Y 397.094,Z 254.018,A -85,B 0,C 180,E1 -11198.276,E2 -11198.276} C_VEL
LIN {X 0,Y 397.055,Z 254.024,A -85,B 0,C 180,E1 -11201.977,E2 -11201.977} C_VEL
LIN {X 0,Y 397.088,Z 254.025,A -85,B 0,C 180,E1 -11205.069,E2 -11205.069} C_VEL
LIN {X 0,Y 397.114,Z 254.108,A -85,B 0,C 180,E1 -11208.589,E2 -11208.589} C_VEL
LIN {X 0,Y 398.038,Z 259.201,A -85,B 0,C 180,E1 -11211.831,E2 -11211.831} C_VEL
LIN {X 0,Y 398.457,Z 263.512,A -85,B 0,C 180,E1 -11214.405,E2 -11214.405} C_VEL
LIN {X 0,Y 398.038,Z 268.904,A -85,B 0,C 180,E1 -11217.417,E2 -11217.417} C_VEL
LIN {X 0,Y 397.51,Z 275.402,A -85,B 0,C 180,E1 -11220.909,E2 -11220.909} C_VEL
LIN {X 0,Y 397.043,Z 282.336,A -85,B 0,C 180,E1 -11224.522,E2 -11224.522} C_VEL
LIN {X 0,Y 396.667,Z 289.431,A -85,B 0,C 180,E1 -11228.156,E2 -11228.156} C_VEL
LIN {X 0,Y 396.309,Z 296.524,A -85,B 0,C 180,E1 -11231.753,E2 -11231.753} C_VEL
LIN {X 0,Y 399.047,Z 310.905,A -85,B 0,C 180,E1 -11232.363,E2 -11232.363} C_VEL
LIN {X 0,Y 400.683,Z 322.979,A -85,B 0,C 180,E1 -11233.037,E2 -11233.037} C_VEL
LIN {X 0,Y 401.049,Z 328.34,A -85,B 0,C 180,E1 -11233.385,E2 -11233.385} C_VEL
LIN {X 0,Y 400.147,Z 339.701,A -85,B 0,C 180,E1 -11234.203,E2 -11234.203} C_VEL
LIN {X 0,Y 399.292,Z 350.679,A -85,B 0,C 180,E1 -11235.213,E2 -11235.213} C_VEL
LIN {X 0,Y 398.51,Z 360.107,A -85,B 0,C 180,E1 -11236.293,E2 -11236.293} C_VEL
LIN {X 0,Y 397.874,Z 368.778,A -85,B 0,C 180,E1 -11237.503,E2 -11237.503} C_VEL
LIN {X 0,Y 397.022,Z 377.714,A -85,B 0,C 180,E1 -11239.03,E2 -11239.03} C_VEL
LIN {X 0,Y 396.504,Z 384.91,A -85,B 0,C 180,E1 -11240.563,E2 -11240.563} C_VEL
LIN {X 0,Y 396.191,Z 389.768,A -85,B 0,C 180,E1 -11241.841,E2 -11241.841} C_VEL
LIN {X 0,Y 395.936,Z 394.492,A -85,B 0,C 180,E1 -11243.375,E2 -11243.375} C_VEL
LIN {X 0,Y 395.845,Z 398.101,A -85,B 0,C 180,E1 -11244.907,E2 -11244.907} C_VEL
LIN {X 0,Y 395.775,Z 399.962,A -85,B 0,C 180,E1 -11245.927,E2 -11245.927} C_VEL
LIN {X 0,Y 395.763,Z 402.355,A -85,B 0,C 180,E1 -11247.965,E2 -11247.965} C_VEL
LIN {X 0,Y 395.791,Z 402.964,A -85,B 0,C 180,E1 -11248.982,E2 -11248.982} C_VEL
LIN {X 0,Y 395.778,Z 403.179,A -85,B 0,C 180,E1 -11250,E2 -11250} C_VEL
LIN {X 0,Y 395.791,Z 402.962,A -85,B 0,C 180,E1 -11251.017,E2 -11251.017} C_VEL
LIN {X 0,Y 395.763,Z 402.352,A -85,B 0,C 180,E1 -11252.035,E2 -11252.035} C_VEL
LIN {X 0,Y 395.775,Z 399.956,A -85,B 0,C 180,E1 -11254.073,E2 -11254.073} C_VEL
LIN {X 0,Y 395.827,Z 396.544,A -85,B 0,C 180,E1 -11255.805,E2 -11255.805} C_VEL
LIN {X 0,Y 396.075,Z 391.441,A -85,B 0,C 180,E1 -11257.648,E2 -11257.648} C_VEL
LIN {X 0,Y 396.428,Z 385.908,A -85,B 0,C 180,E1 -11259.181,E2 -11259.181} C_VEL
LIN {X 0,Y 396.946,Z 379.002,A -85,B 0,C 180,E1 -11260.714,E2 -11260.714} C_VEL
LIN {X 0,Y 397.713,Z 370.366,A -85,B 0,C 180,E1 -11262.243,E2 -11262.243} C_VEL
LIN {X 0,Y 398.456,Z 361.695,A -85,B 0,C 180,E1 -11263.491,E2 -11263.491} C_VEL
LIN {X 0,Y 399.246,Z 351.081,A -85,B 0,C 180,E1 -11264.736,E2 -11264.736} C_VEL
LIN {X 0,Y 400.173,Z 339.611,A -85,B 0,C 180,E1 -11265.796,E2 -11265.796} C_VEL
LIN {X 0,Y 401.003,Z 328.243,A -85,B 0,C 180,E1 -11266.615,E2 -11266.615} C_VEL
LIN {X 0,Y 400.005,Z 317.709,A -85,B 0,C 180,E1 -11267.27,E2 -11267.27} C_VEL
LIN {X 0,Y 397.911,Z 304.535,A -85,B 0,C 180,E1 -11267.921,E2 -11267.921} C_VEL
LIN {X 0,Y 396.307,Z 296.506,A -85,B 0,C 180,E1 -11268.247,E2 -11268.247} C_VEL
LIN {X 0,Y 396.674,Z 289.407,A -85,B 0,C 180,E1 -11271.843,E2 -11271.843} C_VEL
LIN {X 0,Y 397.04,Z 282.312,A -85,B 0,C 180,E1 -11275.478,E2 -11275.478} C_VEL
LIN {X 0,Y 397.516,Z 275.358,A -85,B 0,C 180,E1 -11279.091,E2 -11279.091} C_VEL
LIN {X 0,Y 398.033,Z 268.868,A -85,B 0,C 180,E1 -11282.583,E2 -11282.583} C_VEL
LIN {X 0,Y 398.397,Z 264.551,A -85,B 0,C 180,E1 -11284.982,E2 -11284.982} C_VEL
LIN {X 0,Y 398.173,Z 260.421,A -85,B 0,C 180,E1 -11287.413,E2 -11287.413} C_VEL
LIN {X 0,Y 397.301,Z 254.886,A -85,B 0,C 180,E1 -11290.882,E2 -11290.882} C_VEL
LIN {X 0,Y 397.099,Z 254.024,A -85,B 0,C 180,E1 -11291.582,E2 -11291.582} C_VEL
LIN {X 0,Y 397.087,Z 254.025,A -85,B 0,C 180,E1 -11295.069,E2 -11295.069} C_VEL
LIN {X 0,Y 397.054,Z 254.024,A -85,B 0,C 180,E1 -11298.023,E2 -11298.023} C_VEL
LIN {X 0,Y 397.093,Z 254.019,A -85,B 0,C 180,E1 -11301.724,E2 -11301.724} C_VEL
LIN {X 0,Y 397.126,Z 254.015,A -85,B 0,C 180,E1 -11305.507,E2 -11305.507} C_VEL
LIN {X 0,Y 397.079,Z 254.021,A -85,B 0,C 180,E1 -11309.117,E2 -11309.117} C_VEL
LIN {X 0,Y 397.101,Z 254.02,A -85,B 0,C 180,E1 -11312.603,E2 -11312.603} C_VEL
LIN {X 0,Y 397.113,Z 254.021,A -85,B 0,C 180,E1 -11315.98,E2 -11315.98} C_VEL
LIN {X 0,Y 397.14,Z 254.017,A -85,B 0,C 180,E1 -11319.705,E2 -11319.705} C_VEL
LIN {X 0,Y 397.183,Z 254.008,A -85,B 0,C 180,E1 -11322.845,E2 -11322.845} C_VEL
LIN {X 0,Y 397.23,Z 254.002,A -85,B 0,C 180,E1 -11326.703,E2 -11326.703} C_VEL
LIN {X 0,Y 397.216,Z 254.007,A -85,B 0,C 180,E1 -11329.809,E2 -11329.809} C_VEL
LIN {X 0,Y 397.335,Z 253.99,A -85,B 0,C 180,E1 -11332.888,E2 -11332.888} C_VEL
LIN {X 0,Y 397.253,Z 254.001,A -85,B 0,C 180,E1 -11334.925,E2 -11334.925} C_VEL
LIN {X 0,Y 397.45,Z 253.975,A -85,B 0,C 180,E1 -11337.973,E2 -11337.973} C_VEL
LIN {X 0,Y 397.576,Z 253.959,A -85,B 0,C 180,E1 -11340,E2 -11340} C_VEL
LIN {X 0,Y 397.332,Z 253.993,A -85,B 0,C 180,E1 -11343.042,E2 -11343.042} C_VEL
LIN {X 0,Y 397.325,Z 253.99,A -85,B 0,C 180,E1 -11346.629,E2 -11346.629} C_VEL
LIN {X 0,Y 397.238,Z 254.005,A -85,B 0,C 180,E1 -11349.162,E2 -11349.162} C_VEL
LIN {X 0,Y 397.222,Z 254.005,A -85,B 0,C 180,E1 -11352.258,E2 -11352.258} C_VEL
LIN {X 0,Y 397.18,Z 254.009,A -85,B 0,C 180,E1 -11355.392,E2 -11355.392} C_VEL
LIN {X 0,Y 397.159,Z 254.016,A -85,B 0,C 180,E1 -11358.574,E2 -11358.574} C_VEL
LIN {X 0,Y 397.097,Z 254.018,A -85,B 0,C 180,E1 -11361.819,E2 -11361.819} C_VEL
LIN {X 0,Y 397.154,Z 254.012,A -85,B 0,C 180,E1 -11365.512,E2 -11365.512} C_VEL
LIN {X 0,Y 397.124,Z 254.019,A -85,B 0,C 180,E1 -11368.544,E2 -11368.544} C_VEL
LIN {X 0,Y 397.079,Z 254.025,A -85,B 0,C 180,E1 -11372.072,E2 -11372.072} C_VEL
LIN {X 0,Y 397.1,Z 254.019,A -85,B 0,C 180,E1 -11375.499,E2 -11375.499} C_VEL
LIN {X 0,Y 397.126,Z 254.015,A -85,B 0,C 180,E1 -11378.86,E2 -11378.86} C_VEL
LIN {X 0,Y 397.066,Z 254.025,A -85,B 0,C 180,E1 -11382.268,E2 -11382.268} C_VEL
LIN {X 0,Y 397.085,Z 254.021,A -85,B 0,C 180,E1 -11385.069,E2 -11385.069} C_VEL
LIN {X 0,Y 397.052,Z 254.026,A -85,B 0,C 180,E1 -11388.024,E2 -11388.024} C_VEL
LIN {X 0,Y 397.09,Z 254.022,A -85,B 0,C 180,E1 -11391.724,E2 -11391.724} C_VEL
LIN {X 0,Y 397.012,Z 254.216,A -85,B 0,C 180,E1 -11394.255,E2 -11394.255} C_VEL
LIN {X 0,Y 396.963,Z 257.096,A -85,B 0,C 180,E1 -11396.713,E2 -11396.713} C_VEL
LIN {X 0,Y 396.833,Z 259.974,A -85,B 0,C 180,E1 -11399.096,E2 -11399.096} C_VEL
LIN {X 0,Y 396.639,Z 264.269,A -85,B 0,C 180,E1 -11402.568,E2 -11402.568} C_VEL
LIN {X 0,Y 396.441,Z 268.594,A -85,B 0,C 180,E1 -11405.937,E2 -11405.937} C_VEL
LIN {X 0,Y 396.249,Z 272.957,A -85,B 0,C 180,E1 -11409.223,E2 -11409.223} C_VEL
LIN {X 0,Y 396.17,Z 276.574,A -85,B 0,C 180,E1 -11411.839,E2 -11411.839} C_VEL
LIN {X 0,Y 399.483,Z 290.362,A -85,B 0,C 180,E1 -11412.475,E2 -11412.475} C_VEL
LIN {X 0,Y 401.573,Z 301.486,A -85,B 0,C 180,E1 -11413.136,E2 -11413.136} C_VEL
LIN {X 0,Y 401.102,Z 312.467,A -85,B 0,C 180,E1 -11413.85,E2 -11413.85} C_VEL
LIN {X 0,Y 400.371,Z 323.229,A -85,B 0,C 180,E1 -11414.734,E2 -11414.734} C_VEL
LIN {X 0,Y 399.548,Z 334.196,A -85,B 0,C 180,E1 -11415.874,E2 -11415.874} C_VEL
LIN {X 0,Y 398.621,Z 344.873,A -85,B 0,C 180,E1 -11417.268,E2 -11417.268} C_VEL
LIN {X 0,Y 397.967,Z 352.743,A -85,B 0,C 180,E1 -11418.541,E2 -11418.541} C_VEL
LIN {X 0,Y 397.232,Z 360.438,A -85,B 0,C 180,E1 -11420.067,E2 -11420.067} C_VEL
LIN {X 0,Y 396.736,Z 365.689,A -85,B 0,C 180,E1 -11421.34,E2 -11421.34} C_VEL
LIN {X 0,Y 396.365,Z 370.781,A -85,B 0,C 180,E1 -11422.87,E2 -11422.87} C_VEL
LIN {X 0,Y 396.154,Z 374.734,A -85,B 0,C 180,E1 -11424.401,E2 -11424.401} C_VEL
LIN {X 0,Y 395.888,Z 377.658,A -85,B 0,C 180,E1 -11425.928,E2 -11425.928} C_VEL
LIN {X 0,Y 395.862,Z 379.057,A -85,B 0,C 180,E1 -11426.947,E2 -11426.947} C_VEL
LIN {X 0,Y 395.86,Z 380.051,A -85,B 0,C 180,E1 -11427.965,E2 -11427.965} C_VEL
LIN {X 0,Y 395.779,Z 380.899,A -85,B 0,C 180,E1 -11430,E2 -11430} C_VEL
LIN {X 0,Y 395.797,Z 380.71,A -85,B 0,C 180,E1 -11431.018,E2 -11431.018} C_VEL
LIN {X 0,Y 395.86,Z 380.125,A -85,B 0,C 180,E1 -11432.035,E2 -11432.035} C_VEL
LIN {X 0,Y 395.885,Z 377.806,A -85,B 0,C 180,E1 -11434.072,E2 -11434.072} C_VEL
LIN {X 0,Y 396.133,Z 374.939,A -85,B 0,C 180,E1 -11435.6,E2 -11435.6} C_VEL
LIN {X 0,Y 396.389,Z 371.053,A -85,B 0,C 180,E1 -11437.13,E2 -11437.13} C_VEL
LIN {X 0,Y 396.697,Z 366.042,A -85,B 0,C 180,E1 -11438.661,E2 -11438.661} C_VEL
LIN {X 0,Y 397.279,Z 359.729,A -85,B 0,C 180,E1 -11440.19,E2 -11440.19} C_VEL
LIN {X 0,Y 397.98,Z 351.826,A -85,B 0,C 180,E1 -11441.717,E2 -11441.717} C_VEL
LIN {X 0,Y 398.892,Z 341.993,A -85,B 0,C 180,E1 -11443.241,E2 -11443.241} C_VEL
LIN {X 0,Y 399.723,Z 332.113,A -85,B 0,C 180,E1 -11444.461,E2 -11444.461} C_VEL
LIN {X 0,Y 400.436,Z 321.651,A -85,B 0,C 180,E1 -11445.507,E2 -11445.507} C_VEL
LIN {X 0,Y 400.176,Z 316.652,A -85,B 0,C 180,E1 -11445.958,E2 -11445.958} C_VEL
LIN {X 0,Y 399.04,Z 311.668,A -85,B 0,C 180,E1 -11446.402,E2 -11446.402} C_VEL
LIN {X 0,Y 395.514,Z 301.68,A -85,B 0,C 180,E1 -11447.229,E2 -11447.229} C_VEL
LIN {X 0,Y 393.372,Z 294.682,A -85,B 0,C 180,E1 -11447.714,E2 -11447.714} C_VEL
LIN {X 0,Y 390.351,Z 281.896,A -85,B 0,C 180,E1 -11448.388,E2 -11448.388} C_VEL
LIN {X 0,Y 389.096,Z 276.733,A -85,B 0,C 180,E1 -11448.631,E2 -11448.631} C_VEL
LIN {X 0,Y 389.21,Z 273.28,A -85,B 0,C 180,E1 -11451.171,E2 -11451.171} C_VEL
LIN {X 0,Y 389.383,Z 268.916,A -85,B 0,C 180,E1 -11454.528,E2 -11454.528} C_VEL
LIN {X 0,Y 389.594,Z 264.566,A -85,B 0,C 180,E1 -11457.971,E2 -11457.971} C_VEL
LIN {X 0,Y 389.77,Z 260.239,A -85,B 0,C 180,E1 -11461.527,E2 -11461.527} C_VEL
LIN {X 0,Y 389.922,Z 257.345,A -85,B 0,C 180,E1 -11463.992,E2 -11463.992} C_VEL
LIN {X 0,Y 389.958,Z 255.253,A -85,B 0,C 180,E1 -11465.805,E2 -11465.805} C_VEL
LIN {X 0,Y 389.969,Z 254.911,A -85,B 0,C 180,E1 -11466.493,E2 -11466.493} C_VEL
LIN {X 0,Y 390.039,Z 254.898,A -85,B 0,C 180,E1 -11469.212,E2 -11469.212} C_VEL
LIN {X 0,Y 390.032,Z 254.904,A -85,B 0,C 180,E1 -11472.372,E2 -11472.372} C_VEL
LIN {X 0,Y 390.045,Z 254.897,A -85,B 0,C 180,E1 -11475.354,E2 -11475.354} C_VEL
LIN {X 0,Y 390.027,Z 254.904,A -85,B 0,C 180,E1 -11478.186,E2 -11478.186} C_VEL
LIN {X 0,Y 390.089,Z 254.892,A -85,B 0,C 180,E1 -11480.907,E2 -11480.907} C_VEL
LIN {X 0,Y 390.087,Z 254.891,A -85,B 0,C 180,E1 -11484.793,E2 -11484.793} C_VEL
LIN {X 0,Y 390.026,Z 254.9,A -85,B 0,C 180,E1 -11488.496,E2 -11488.496} C_VEL
LIN {X 0,Y 390.12,Z 254.891,A -85,B 0,C 180,E1 -11492.07,E2 -11492.07} C_VEL
LIN {X 0,Y 390.08,Z 254.897,A -85,B 0,C 180,E1 -11495.519,E2 -11495.519} C_VEL
LIN {X 0,Y 390.09,Z 254.897,A -85,B 0,C 180,E1 -11499.53,E2 -11499.53} C_VEL
LIN {X 0,Y 390.14,Z 254.89,A -85,B 0,C 180,E1 -11503.248,E2 -11503.248} C_VEL
LIN {X 0,Y 390.198,Z 254.878,A -85,B 0,C 180,E1 -11506.562,E2 -11506.562} C_VEL
LIN {X 0,Y 390.171,Z 254.883,A -85,B 0,C 180,E1 -11509.623,E2 -11509.623} C_VEL
LIN {X 0,Y 390.282,Z 254.87,A -85,B 0,C 180,E1 -11512.758,E2 -11512.758} C_VEL
LIN {X 0,Y 390.215,Z 254.88,A -85,B 0,C 180,E1 -11514.833,E2 -11514.833} C_VEL
LIN {X 0,Y 390.413,Z 254.851,A -85,B 0,C 180,E1 -11517.937,E2 -11517.937} C_VEL
LIN {X 0,Y 390.343,Z 254.864,A -85,B 0,C 180,E1 -11521.032,E2 -11521.032} C_VEL
LIN {X 0,Y 390.312,Z 254.866,A -85,B 0,C 180,E1 -11523.096,E2 -11523.096} C_VEL
LIN {X 0,Y 390.32,Z 254.865,A -85,B 0,C 180,E1 -11526.202,E2 -11526.202} C_VEL
LIN {X 0,Y 390.19,Z 254.878,A -85,B 0,C 180,E1 -11529.329,E2 -11529.329} C_VEL
LIN {X 0,Y 390.197,Z 254.878,A -85,B 0,C 180,E1 -11533.438,E2 -11533.438} C_VEL
LIN {X 0,Y 390.152,Z 254.884,A -85,B 0,C 180,E1 -11537.308,E2 -11537.308} C_VEL
LIN {X 0,Y 390.09,Z 254.894,A -85,B 0,C 180,E1 -11540.47,E2 -11540.47} C_VEL
LIN {X 0,Y 390.064,Z 254.895,A -85,B 0,C 180,E1 -11543.352,E2 -11543.352} C_VEL
LIN {X 0,Y 390.053,Z 254.896,A -85,B 0,C 180,E1 -11546.773,E2 -11546.773} C_VEL
LIN {X 0,Y 390.039,Z 254.899,A -85,B 0,C 180,E1 -11550.3,E2 -11550.3} C_VEL
LIN {X 0,Y 390.07,Z 254.896,A -85,B 0,C 180,E1 -11554.024,E2 -11554.024} C_VEL
LIN {X 0,Y 390.041,Z 254.903,A -85,B 0,C 180,E1 -11557.55,E2 -11557.55} C_VEL
LIN {X 0,Y 390.019,Z 254.901,A -85,B 0,C 180,E1 -11560.815,E2 -11560.815} C_VEL
LIN {X 0,Y 390.054,Z 254.899,A -85,B 0,C 180,E1 -11563.886,E2 -11563.886} C_VEL
LIN {X 0,Y 390.06,Z 254.9,A -85,B 0,C 180,E1 -11566.79,E2 -11566.79} C_VEL
LIN {X 0,Y 390.063,Z 255.011,A -85,B 0,C 180,E1 -11568.318,E2 -11568.318} C_VEL
LIN {X 0,Y 390.832,Z 259.099,A -85,B 0,C 180,E1 -11570.996,E2 -11570.996} C_VEL
LIN {X 0,Y 391.375,Z 263.817,A -85,B 0,C 180,E1 -11573.908,E2 -11573.908} C_VEL
LIN {X 0,Y 391.21,Z 267.695,A -85,B 0,C 180,E1 -11576.158,E2 -11576.158} C_VEL
LIN {X 0,Y 390.657,Z 274.174,A -85,B 0,C 180,E1 -11579.753,E2 -11579.753} C_VEL
LIN {X 0,Y 390.157,Z 280.672,A -85,B 0,C 180,E1 -11583.235,E2 -11583.235} C_VEL
LIN {X 0,Y 389.727,Z 287.595,A -85,B 0,C 180,E1 -11586.881,E2 -11586.881} C_VEL
LIN {X 0,Y 389.425,Z 293.498,A -85,B 0,C 180,E1 -11589.946,E2 -11589.946} C_VEL
LIN {X 0,Y 389.262,Z 296.505,A -85,B 0,C 180,E1 -11591.428,E2 -11591.428} C_VEL
LIN {X 0,Y 391.853,Z 309.567,A -85,B 0,C 180,E1 -11591.978,E2 -11591.978} C_VEL
LIN {X 0,Y 393.53,Z 321.58,A -85,B 0,C 180,E1 -11592.649,E2 -11592.649} C_VEL
LIN {X 0,Y 394.12,Z 330.005,A -85,B 0,C 180,E1 -11593.209,E2 -11593.209} C_VEL
LIN {X 0,Y 393.178,Z 341.04,A -85,B 0,C 180,E1 -11594.048,E2 -11594.048} C_VEL
LIN {X 0,Y 392.196,Z 352.836,A -85,B 0,C 180,E1 -11595.205,E2 -11595.205} C_VEL
LIN {X 0,Y 391.341,Z 363.316,A -85,B 0,C 180,E1 -11596.499,E2 -11596.499} C_VEL
LIN {X 0,Y 390.63,Z 371.798,A -85,B 0,C 180,E1 -11597.795,E2 -11597.795} C_VEL
LIN {X 0,Y 389.852,Z 380.075,A -85,B 0,C 180,E1 -11599.352,E2 -11599.352} C_VEL
LIN {X 0,Y 389.339,Z 386.749,A -85,B 0,C 180,E1 -11600.912,E2 -11600.912} C_VEL
LIN {X 0,Y 388.938,Z 392.858,A -85,B 0,C 180,E1 -11602.733,E2 -11602.733} C_VEL
LIN {X 0,Y 388.731,Z 396.714,A -85,B 0,C 180,E1 -11604.24,E2 -11604.24} C_VEL
LIN {X 0,Y 388.7,Z 399.763,A -85,B 0,C 180,E1 -11605.852,E2 -11605.852} C_VEL
LIN {X 0,Y 388.661,Z 402.156,A -85,B 0,C 180,E1 -11607.927,E2 -11607.927} C_VEL
LIN {X 0,Y 388.703,Z 402.765,A -85,B 0,C 180,E1 -11608.964,E2 -11608.964} C_VEL
LIN {X 0,Y 388.707,Z 402.98,A -85,B 0,C 180,E1 -11610,E2 -11610} C_VEL
LIN {X 0,Y 388.703,Z 402.762,A -85,B 0,C 180,E1 -11611.036,E2 -11611.036} C_VEL
LIN {X 0,Y 388.661,Z 402.152,A -85,B 0,C 180,E1 -11612.072,E2 -11612.072} C_VEL
LIN {X 0,Y 388.7,Z 399.755,A -85,B 0,C 180,E1 -11614.147,E2 -11614.147} C_VEL
LIN {X 0,Y 388.727,Z 396.713,A -85,B 0,C 180,E1 -11615.754,E2 -11615.754} C_VEL
LIN {X 0,Y 388.937,Z 392.836,A -85,B 0,C 180,E1 -11617.267,E2 -11617.267} C_VEL
LIN {X 0,Y 389.339,Z 386.719,A -85,B 0,C 180,E1 -11619.088,E2 -11619.088} C_VEL
LIN {X 0,Y 389.852,Z 380.038,A -85,B 0,C 180,E1 -11620.648,E2 -11620.648} C_VEL
LIN {X 0,Y 390.619,Z 371.752,A -85,B 0,C 180,E1 -11622.205,E2 -11622.205} C_VEL
LIN {X 0,Y 391.355,Z 363.257,A -85,B 0,C 180,E1 -11623.501,E2 -11623.501} C_VEL
LIN {X 0,Y 392.196,Z 352.761,A -85,B 0,C 180,E1 -11624.795,E2 -11624.795} C_VEL
LIN {X 0,Y 393.084,Z 342.38,A -85,B 0,C 180,E1 -11625.822,E2 -11625.822} C_VEL
LIN {X 0,Y 393.973,Z 331.365,A -85,B 0,C 180,E1 -11626.69,E2 -11626.69} C_VEL
LIN {X 0,Y 394.056,Z 326.721,A -85,B 0,C 180,E1 -11627.004,E2 -11627.004} C_VEL
LIN {X 0,Y 392.504,Z 314.088,A -85,B 0,C 180,E1 -11627.782,E2 -11627.782} C_VEL
LIN {X 0,Y 390.482,Z 302.49,A -85,B 0,C 180,E1 -11628.334,E2 -11628.334} C_VEL
LIN {X 0,Y 389.253,Z 296.313,A -85,B 0,C 180,E1 -11628.589,E2 -11628.589} C_VEL
LIN {X 0,Y 389.664,Z 289.227,A -85,B 0,C 180,E1 -11632.257,E2 -11632.257} C_VEL
LIN {X 0,Y 390.008,Z 282.632,A -85,B 0,C 180,E1 -11635.709,E2 -11635.709} C_VEL
LIN {X 0,Y 390.576,Z 275.214,A -85,B 0,C 180,E1 -11639.659,E2 -11639.659} C_VEL
LIN {X 0,Y 391.137,Z 268.725,A -85,B 0,C 180,E1 -11643.232,E2 -11643.232} C_VEL
LIN {X 0,Y 391.377,Z 265.491,A -85,B 0,C 180,E1 -11645.074,E2 -11645.074} C_VEL
LIN {X 0,Y 391.094,Z 261.056,A -85,B 0,C 180,E1 -11647.75,E2 -11647.75} C_VEL
LIN {X 0,Y 390.334,Z 256.182,A -85,B 0,C 180,E1 -11650.868,E2 -11650.868} C_VEL
LIN {X 0,Y 390.051,Z 254.902,A -85,B 0,C 180,E1 -11651.811,E2 -11651.811} C_VEL
LIN {X 0,Y 390.044,Z 254.902,A -85,B 0,C 180,E1 -11655.354,E2 -11655.354} C_VEL
LIN {X 0,Y 390.017,Z 254.902,A -85,B 0,C 180,E1 -11658.185,E2 -11658.185} C_VEL
LIN {X 0,Y 390.058,Z 254.898,A -85,B 0,C 180,E1 -11660.904,E2 -11660.904} C_VEL
LIN {X 0,Y 390.086,Z 254.895,A -85,B 0,C 180,E1 -11664.793,E2 -11664.793} C_VEL
LIN {X 0,Y 390.025,Z 254.904,A -85,B 0,C 180,E1 -11668.496,E2 -11668.496} C_VEL
LIN {X 0,Y 390.038,Z 254.902,A -85,B 0,C 180,E1 -11672.064,E2 -11672.064} C_VEL
LIN {X 0,Y 390.044,Z 254.898,A -85,B 0,C 180,E1 -11675.517,E2 -11675.517} C_VEL
LIN {X 0,Y 390.056,Z 254.895,A -85,B 0,C 180,E1 -11678.878,E2 -11678.878} C_VEL
LIN {X 0,Y 390.13,Z 254.89,A -85,B 0,C 180,E1 -11682.167,E2 -11682.167} C_VEL
LIN {X 0,Y 390.145,Z 254.887,A -85,B 0,C 180,E1 -11685.393,E2 -11685.393} C_VEL
LIN {X 0,Y 390.146,Z 254.884,A -85,B 0,C 180,E1 -11688.571,E2 -11688.571} C_VEL
LIN {X 0,Y 390.271,Z 254.87,A -85,B 0,C 180,E1 -11692.071,E2 -11692.071} C_VEL
LIN {X 0,Y 390.225,Z 254.876,A -85,B 0,C 180,E1 -11694.834,E2 -11694.834} C_VEL
LIN {X 0,Y 390.419,Z 254.851,A -85,B 0,C 180,E1 -11697.937,E2 -11697.937} C_VEL
LIN {X 0,Y 390.545,Z 254.835,A -85,B 0,C 180,E1 -11700,E2 -11700} C_VEL
LIN {X 0,Y 390.269,Z 254.874,A -85,B 0,C 180,E1 -11703.097,E2 -11703.097} C_VEL
LIN {X 0,Y 390.28,Z 254.867,A -85,B 0,C 180,E1 -11706.624,E2 -11706.624} C_VEL
LIN {X 0,Y 390.195,Z 254.88,A -85,B 0,C 180,E1 -11709.329,E2 -11709.329} C_VEL
LIN {X 0,Y 390.173,Z 254.884,A -85,B 0,C 180,E1 -11712.483,E2 -11712.483} C_VEL
LIN {X 0,Y 390.14,Z 254.885,A -85,B 0,C 180,E1 -11715.677,E2 -11715.677} C_VEL
LIN {X 0,Y 390.104,Z 254.892,A -85,B 0,C 180,E1 -11718.922,E2 -11718.922} C_VEL
LIN {X 0,Y 390.039,Z 254.901,A -85,B 0,C 180,E1 -11722.234,E2 -11722.234} C_VEL
LIN {X 0,Y 390.12,Z 254.888,A -85,B 0,C 180,E1 -11725.743,E2 -11725.743} C_VEL
LIN {X 0,Y 390.06,Z 254.895,A -85,B 0,C 180,E1 -11729.11,E2 -11729.11} C_VEL
LIN {X 0,Y 390.042,Z 254.898,A -85,B 0,C 180,E1 -11732.722,E2 -11732.722} C_VEL
LIN {X 0,Y 390.045,Z 254.901,A -85,B 0,C 180,E1 -11735.823,E2 -11735.823} C_VEL
LIN {X 0,Y 390.062,Z 254.895,A -85,B 0,C 180,E1 -11739.217,E2 -11739.217} C_VEL
LIN {X 0,Y 390.04,Z 254.899,A -85,B 0,C 180,E1 -11742.374,E2 -11742.374} C_VEL
LIN {X 0,Y 390.041,Z 254.9,A -85,B 0,C 180,E1 -11745.354,E2 -11745.354} C_VEL
LIN {X 0,Y 390.015,Z 254.901,A -85,B 0,C 180,E1 -11748.185,E2 -11748.185} C_VEL
LIN {X 0,Y 390.059,Z 254.895,A -85,B 0,C 180,E1 -11750.904,E2 -11750.904} C_VEL
LIN {X 0,Y 389.969,Z 255.112,A -85,B 0,C 180,E1 -11754.193,E2 -11754.193} C_VEL
LIN {X 0,Y 389.877,Z 258.694,A -85,B 0,C 180,E1 -11757.263,E2 -11757.263} C_VEL
LIN {X 0,Y 389.67,Z 262.997,A -85,B 0,C 180,E1 -11760.859,E2 -11760.859} C_VEL
LIN {X 0,Y 389.456,Z 267.472,A -85,B 0,C 180,E1 -11764.461,E2 -11764.461} C_VEL
LIN {X 0,Y 389.265,Z 271.686,A -85,B 0,C 180,E1 -11767.719,E2 -11767.719} C_VEL
LIN {X 0,Y 389.106,Z 276.13,A -85,B 0,C 180,E1 -11771.028,E2 -11771.028} C_VEL
LIN {X 0,Y 389.091,Z 276.773,A -85,B 0,C 180,E1 -11771.498,E2 -11771.498} C_VEL
LIN {X 0,Y 392.33,Z 289.867,A -85,B 0,C 180,E1 -11772.113,E2 -11772.113} C_VEL
LIN {X 0,Y 394.731,Z 302.306,A -85,B 0,C 180,E1 -11772.871,E2 -11772.871} C_VEL
LIN {X 0,Y 394.304,Z 312.672,A -85,B 0,C 180,E1 -11773.564,E2 -11773.564} C_VEL
LIN {X 0,Y 393.545,Z 323.433,A -85,B 0,C 180,E1 -11774.462,E2 -11774.462} C_VEL
LIN {X 0,Y 392.663,Z 334.4,A -85,B 0,C 180,E1 -11775.621,E2 -11775.621} C_VEL
LIN {X 0,Y 391.869,Z 343.302,A -85,B 0,C 180,E1 -11776.782,E2 -11776.782} C_VEL
LIN {X 0,Y 391.099,Z 351.469,A -85,B 0,C 180,E1 -11778.074,E2 -11778.074} C_VEL
LIN {X 0,Y 390.326,Z 359.469,A -85,B 0,C 180,E1 -11779.627,E2 -11779.627} C_VEL
LIN {X 0,Y 389.716,Z 365.891,A -85,B 0,C 180,E1 -11781.183,E2 -11781.183} C_VEL
LIN {X 0,Y 389.317,Z 370.983,A -85,B 0,C 180,E1 -11782.74,E2 -11782.74} C_VEL
LIN {X 0,Y 389.087,Z 374.935,A -85,B 0,C 180,E1 -11784.299,E2 -11784.299} C_VEL
LIN {X 0,Y 388.815,Z 377.858,A -85,B 0,C 180,E1 -11785.854,E2 -11785.854} C_VEL
LIN {X 0,Y 388.767,Z 379.257,A -85,B 0,C 180,E1 -11786.891,E2 -11786.891} C_VEL
LIN {X 0,Y 388.762,Z 380.251,A -85,B 0,C 180,E1 -11787.928,E2 -11787.928} C_VEL
LIN {X 0,Y 388.708,Z 381.098,A -85,B 0,C 180,E1 -11790,E2 -11790} C_VEL
LIN {X 0,Y 388.728,Z 380.909,A -85,B 0,C 180,E1 -11791.036,E2 -11791.036} C_VEL
LIN {X 0,Y 388.762,Z 380.325,A -85,B 0,C 180,E1 -11792.072,E2 -11792.072} C_VEL
LIN {X 0,Y 388.811,Z 378.005,A -85,B 0,C 180,E1 -11794.146,E2 -11794.146} C_VEL
LIN {X 0,Y 389.07,Z 375.137,A -85,B 0,C 180,E1 -11795.702,E2 -11795.702} C_VEL
LIN {X 0,Y 389.333,Z 371.252,A -85,B 0,C 180,E1 -11797.259,E2 -11797.259} C_VEL
LIN {X 0,Y 389.679,Z 366.24,A -85,B 0,C 180,E1 -11798.818,E2 -11798.818} C_VEL
LIN {X 0,Y 390.294,Z 359.927,A -85,B 0,C 180,E1 -11800.374,E2 -11800.374} C_VEL
LIN {X 0,Y 391.024,Z 352.024,A -85,B 0,C 180,E1 -11801.929,E2 -11801.929} C_VEL
LIN {X 0,Y 391.973,Z 342.19,A -85,B 0,C 180,E1 -11803.479,E2 -11803.479} C_VEL
LIN {X 0,Y 392.811,Z 332.657,A -85,B 0,C 180,E1 -11804.682,E2 -11804.682} C_VEL
LIN {X 0,Y 393.6,Z 321.649,A -85,B 0,C 180,E1 -11805.801,E2 -11805.801} C_VEL
LIN {X 0,Y 394.603,Z 309.417,A -85,B 0,C 180,E1 -11806.768,E2 -11806.768} C_VEL
LIN {X 0,Y 394.876,Z 303.03,A -85,B 0,C 180,E1 -11807.179,E2 -11807.179} C_VEL
LIN {X 0,Y 393.372,Z 294.682,A -85,B 0,C 180,E1 -11807.714,E2 -11807.714} C_VEL
LIN {X 0,Y 391.934,Z 291.334,A -85,B 0,C 180,E1 -11807.947,E2 -11807.947} C_VEL
LIN {X 0,Y 388.008,Z 286.575,A -85,B 0,C 180,E1 -11808.342,E2 -11808.342} C_VEL
LIN {X 0,Y 383.956,Z 281.78,A -85,B 0,C 180,E1 -11808.715,E2 -11808.715} C_VEL
LIN {X 0,Y 382.3,Z 278.366,A -85,B 0,C 180,E1 -11808.904,E2 -11808.904} C_VEL
LIN {X 0,Y 382.042,Z 276.929,A -85,B 0,C 180,E1 -11808.988,E2 -11808.988} C_VEL
LIN {X 0,Y 382.146,Z 273.467,A -85,B 0,C 180,E1 -11811.581,E2 -11811.581} C_VEL
LIN {X 0,Y 382.344,Z 269.084,A -85,B 0,C 180,E1 -11815.01,E2 -11815.01} C_VEL
LIN {X 0,Y 382.564,Z 264.718,A -85,B 0,C 180,E1 -11818.532,E2 -11818.532} C_VEL
LIN {X 0,Y 382.769,Z 260.401,A -85,B 0,C 180,E1 -11822.173,E2 -11822.173} C_VEL
LIN {X 0,Y 382.897,Z 257.504,A -85,B 0,C 180,E1 -11824.681,E2 -11824.681} C_VEL
LIN {X 0,Y 382.921,Z 255.849,A -85,B 0,C 180,E1 -11826.141,E2 -11826.141} C_VEL
LIN {X 0,Y 382.981,Z 255.782,A -85,B 0,C 180,E1 -11828.604,E2 -11828.604} C_VEL
LIN {X 0,Y 382.962,Z 255.779,A -85,B 0,C 180,E1 -11831.351,E2 -11831.351} C_VEL
LIN {X 0,Y 382.991,Z 255.781,A -85,B 0,C 180,E1 -11834.302,E2 -11834.302} C_VEL
LIN {X 0,Y 383.013,Z 255.773,A -85,B 0,C 180,E1 -11837.24,E2 -11837.24} C_VEL
LIN {X 0,Y 383.01,Z 255.777,A -85,B 0,C 180,E1 -11840.415,E2 -11840.415} C_VEL
LIN {X 0,Y 383.027,Z 255.776,A -85,B 0,C 180,E1 -11844.044,E2 -11844.044} C_VEL
LIN {X 0,Y 382.989,Z 255.778,A -85,B 0,C 180,E1 -11847.578,E2 -11847.578} C_VEL
LIN {X 0,Y 382.994,Z 255.777,A -85,B 0,C 180,E1 -11850.3,E2 -11850.3} C_VEL
LIN {X 0,Y 383.059,Z 255.767,A -85,B 0,C 180,E1 -11852.698,E2 -11852.698} C_VEL
LIN {X 0,Y 383.054,Z 255.768,A -85,B 0,C 180,E1 -11855.04,E2 -11855.04} C_VEL
LIN {X 0,Y 382.995,Z 255.774,A -85,B 0,C 180,E1 -11858.469,E2 -11858.469} C_VEL
LIN {X 0,Y 383.055,Z 255.77,A -85,B 0,C 180,E1 -11861.826,E2 -11861.826} C_VEL
LIN {X 0,Y 383.111,Z 255.765,A -85,B 0,C 180,E1 -11865.118,E2 -11865.118} C_VEL
LIN {X 0,Y 383.1,Z 255.762,A -85,B 0,C 180,E1 -11868.358,E2 -11868.358} C_VEL
LIN {X 0,Y 383.23,Z 255.745,A -85,B 0,C 180,E1 -11872.014,E2 -11872.014} C_VEL
LIN {X 0,Y 383.187,Z 255.754,A -85,B 0,C 180,E1 -11874.738,E2 -11874.738} C_VEL
LIN {X 0,Y 383.379,Z 255.727,A -85,B 0,C 180,E1 -11877.899,E2 -11877.899} C_VEL
LIN {X 0,Y 383.309,Z 255.739,A -85,B 0,C 180,E1 -11881.051,E2 -11881.051} C_VEL
LIN {X 0,Y 383.249,Z 255.745,A -85,B 0,C 180,E1 -11883.154,E2 -11883.154} C_VEL
LIN {X 0,Y 383.275,Z 255.743,A -85,B 0,C 180,E1 -11886.316,E2 -11886.316} C_VEL
LIN {X 0,Y 383.14,Z 255.756,A -85,B 0,C 180,E1 -11889.502,E2 -11889.502} C_VEL
LIN {X 0,Y 383.128,Z 255.758,A -85,B 0,C 180,E1 -11893.536,E2 -11893.536} C_VEL
LIN {X 0,Y 383.098,Z 255.763,A -85,B 0,C 180,E1 -11897.455,E2 -11897.455} C_VEL
LIN {X 0,Y 383.031,Z 255.771,A -85,B 0,C 180,E1 -11900.647,E2 -11900.647} C_VEL
LIN {X 0,Y 383.012,Z 255.777,A -85,B 0,C 180,E1 -11903.809,E2 -11903.809} C_VEL
LIN {X 0,Y 382.993,Z 255.776,A -85,B 0,C 180,E1 -11907.307,E2 -11907.307} C_VEL
LIN {X 0,Y 382.984,Z 255.776,A -85,B 0,C 180,E1 -11910.919,E2 -11910.919} C_VEL
LIN {X 0,Y 383.02,Z 255.772,A -85,B 0,C 180,E1 -11914.668,E2 -11914.668} C_VEL
LIN {X 0,Y 382.995,Z 255.777,A -85,B 0,C 180,E1 -11917.902,E2 -11917.902} C_VEL
LIN {X 0,Y 382.963,Z 255.784,A -85,B 0,C 180,E1 -11921.35,E2 -11921.35} C_VEL
LIN {X 0,Y 382.996,Z 255.779,A -85,B 0,C 180,E1 -11924.303,E2 -11924.303} C_VEL
LIN {X 0,Y 383.028,Z 255.901,A -85,B 0,C 180,E1 -11928.043,E2 -11928.043} C_VEL
LIN {X 0,Y 383.955,Z 261.12,A -85,B 0,C 180,E1 -11931.512,E2 -11931.512} C_VEL
LIN {X 0,Y 384.315,Z 264.407,A -85,B 0,C 180,E1 -11933.575,E2 -11933.575} C_VEL
LIN {X 0,Y 384.293,Z 267.577,A -85,B 0,C 180,E1 -11935.463,E2 -11935.463} C_VEL
LIN {X 0,Y 383.821,Z 272.952,A -85,B 0,C 180,E1 -11938.543,E2 -11938.543} C_VEL
LIN {X 0,Y 383.288,Z 278.583,A -85,B 0,C 180,E1 -11941.658,E2 -11941.658} C_VEL
LIN {X 0,Y 382.866,Z 284.793,A -85,B 0,C 180,E1 -11945.027,E2 -11945.027} C_VEL
LIN {X 0,Y 382.518,Z 291.203,A -85,B 0,C 180,E1 -11948.441,E2 -11948.441} C_VEL
LIN {X 0,Y 382.201,Z 296.313,A -85,B 0,C 180,E1 -11951.072,E2 -11951.072} C_VEL
LIN {X 0,Y 384.804,Z 309.254,A -85,B 0,C 180,E1 -11951.631,E2 -11951.631} C_VEL
LIN {X 0,Y 386.495,Z 320.93,A -85,B 0,C 180,E1 -11952.295,E2 -11952.295} C_VEL
LIN {X 0,Y 387.299,Z 329.969,A -85,B 0,C 180,E1 -11952.915,E2 -11952.915} C_VEL
LIN {X 0,Y 386.231,Z 342.273,A -85,B 0,C 180,E1 -11953.889,E2 -11953.889} C_VEL
LIN {X 0,Y 385.213,Z 353.816,A -85,B 0,C 180,E1 -11955.066,E2 -11955.066} C_VEL
LIN {X 0,Y 384.395,Z 363.117,A -85,B 0,C 180,E1 -11956.25,E2 -11956.25} C_VEL
LIN {X 0,Y 383.659,Z 371.599,A -85,B 0,C 180,E1 -11957.57,E2 -11957.57} C_VEL
LIN {X 0,Y 382.825,Z 379.875,A -85,B 0,C 180,E1 -11959.154,E2 -11959.154} C_VEL
LIN {X 0,Y 382.276,Z 386.549,A -85,B 0,C 180,E1 -11960.743,E2 -11960.743} C_VEL
LIN {X 0,Y 381.866,Z 392.658,A -85,B 0,C 180,E1 -11962.598,E2 -11962.598} C_VEL
LIN {X 0,Y 381.689,Z 395.927,A -85,B 0,C 180,E1 -11963.879,E2 -11963.879} C_VEL
LIN {X 0,Y 381.625,Z 399.564,A -85,B 0,C 180,E1 -11965.775,E2 -11965.775} C_VEL
LIN {X 0,Y 381.56,Z 401.956,A -85,B 0,C 180,E1 -11967.889,E2 -11967.889} C_VEL
LIN {X 0,Y 381.617,Z 402.566,A -85,B 0,C 180,E1 -11968.945,E2 -11968.945} C_VEL
LIN {X 0,Y 381.639,Z 402.781,A -85,B 0,C 180,E1 -11970,E2 -11970} C_VEL
LIN {X 0,Y 381.617,Z 402.563,A -85,B 0,C 180,E1 -11971.055,E2 -11971.055} C_VEL
LIN {X 0,Y 381.546,Z 400.953,A -85,B 0,C 180,E1 -11973.168,E2 -11973.168} C_VEL
LIN {X 0,Y 381.625,Z 399.555,A -85,B 0,C 180,E1 -11974.224,E2 -11974.224} C_VEL
LIN {X 0,Y 381.687,Z 395.913,A -85,B 0,C 180,E1 -11976.118,E2 -11976.118} C_VEL
LIN {X 0,Y 381.953,Z 391.038,A -85,B 0,C 180,E1 -11977.932,E2 -11977.932} C_VEL
LIN {X 0,Y 382.373,Z 385.504,A -85,B 0,C 180,E1 -11979.522,E2 -11979.522} C_VEL
LIN {X 0,Y 382.909,Z 378.597,A -85,B 0,C 180,E1 -11981.111,E2 -11981.111} C_VEL
LIN {X 0,Y 383.809,Z 369.96,A -85,B 0,C 180,E1 -11982.693,E2 -11982.693} C_VEL
LIN {X 0,Y 384.67,Z 360.256,A -85,B 0,C 180,E1 -11984.126,E2 -11984.126} C_VEL
LIN {X 0,Y 385.543,Z 350.202,A -85,B 0,C 180,E1 -11985.326,E2 -11985.326} C_VEL
LIN {X 0,Y 386.498,Z 339.202,A -85,B 0,C 180,E1 -11986.371,E2 -11986.371} C_VEL
LIN {X 0,Y 387.245,Z 328.349,A -85,B 0,C 180,E1 -11987.187,E2 -11987.187} C_VEL
LIN {X 0,Y 385.849,Z 316.2,A -85,B 0,C 180,E1 -11987.981,E2 -11987.981} C_VEL
LIN {X 0,Y 383.842,Z 304.273,A -85,B 0,C 180,E1 -11988.595,E2 -11988.595} C_VEL
LIN {X 0,Y 382.197,Z 296.103,A -85,B 0,C 180,E1 -11988.946,E2 -11988.946} C_VEL
LIN {X 0,Y 382.569,Z 290.118,A -85,B 0,C 180,E1 -11992.123,E2 -11992.123} C_VEL
LIN {X 0,Y 382.991,Z 282.952,A -85,B 0,C 180,E1 -11995.951,E2 -11995.951} C_VEL
LIN {X 0,Y 383.536,Z 276.154,A -85,B 0,C 180,E1 -11999.654,E2 -11999.654} C_VEL
LIN {X 0,Y 384.114,Z 269.67,A -85,B 0,C 180,E1 -12003.292,E2 -12003.292} C_VEL
LIN {X 0,Y 384.346,Z 265.374,A -85,B 0,C 180,E1 -12005.813,E2 -12005.813} C_VEL
LIN {X 0,Y 384.003,Z 261.705,A -85,B 0,C 180,E1 -12008.095,E2 -12008.095} C_VEL
LIN {X 0,Y 383.216,Z 256.799,A -85,B 0,C 180,E1 -12011.317,E2 -12011.317} C_VEL
LIN {X 0,Y 383.001,Z 255.781,A -85,B 0,C 180,E1 -12012.049,E2 -12012.049} C_VEL
LIN {X 0,Y 382.996,Z 255.778,A -85,B 0,C 180,E1 -12015.789,E2 -12015.789} C_VEL
LIN {X 0,Y 382.962,Z 255.783,A -85,B 0,C 180,E1 -12018.8,E2 -12018.8} C_VEL
LIN {X 0,Y 382.994,Z 255.777,A -85,B 0,C 180,E1 -12022.097,E2 -12022.097} C_VEL
LIN {X 0,Y 383.019,Z 255.772,A -85,B 0,C 180,E1 -12025.332,E2 -12025.332} C_VEL
LIN {X 0,Y 382.983,Z 255.777,A -85,B 0,C 180,E1 -12029.081,E2 -12029.081} C_VEL
LIN {X 0,Y 382.992,Z 255.776,A -85,B 0,C 180,E1 -12032.693,E2 -12032.693} C_VEL
LIN {X 0,Y 383.011,Z 255.777,A -85,B 0,C 180,E1 -12036.191,E2 -12036.191} C_VEL
LIN {X 0,Y 383.057,Z 255.77,A -85,B 0,C 180,E1 -12039.599,E2 -12039.599} C_VEL
LIN {X 0,Y 383.107,Z 255.761,A -85,B 0,C 180,E1 -12042.931,E2 -12042.931} C_VEL
LIN {X 0,Y 383.127,Z 255.759,A -85,B 0,C 180,E1 -12046.464,E2 -12046.464} C_VEL
LIN {X 0,Y 383.143,Z 255.756,A -85,B 0,C 180,E1 -12050.498,E2 -12050.498} C_VEL
LIN {X 0,Y 383.274,Z 255.744,A -85,B 0,C 180,E1 -12053.684,E2 -12053.684} C_VEL
LIN {X 0,Y 383.387,Z 255.727,A -85,B 0,C 180,E1 -12057.899,E2 -12057.899} C_VEL
LIN {X 0,Y 383.515,Z 255.71,A -85,B 0,C 180,E1 -12060,E2 -12060} C_VEL
LIN {X 0,Y 383.207,Z 255.754,A -85,B 0,C 180,E1 -12063.154,E2 -12063.154} C_VEL
LIN {X 0,Y 383.24,Z 255.743,A -85,B 0,C 180,E1 -12066.615,E2 -12066.615} C_VEL
LIN {X 0,Y 383.146,Z 255.757,A -85,B 0,C 180,E1 -12069.502,E2 -12069.502} C_VEL
LIN {X 0,Y 383.138,Z 255.762,A -85,B 0,C 180,E1 -12072.716,E2 -12072.716} C_VEL
LIN {X 0,Y 383.082,Z 255.764,A -85,B 0,C 180,E1 -12075.973,E2 -12075.973} C_VEL
LIN {X 0,Y 383.06,Z 255.767,A -85,B 0,C 180,E1 -12079.284,E2 -12079.284} C_VEL
LIN {X 0,Y 382.993,Z 255.779,A -85,B 0,C 180,E1 -12082.666,E2 -12082.666} C_VEL
LIN {X 0,Y 383.081,Z 255.768,A -85,B 0,C 180,E1 -12086.123,E2 -12086.123} C_VEL
LIN {X 0,Y 383.042,Z 255.773,A -85,B 0,C 180,E1 -12088.493,E2 -12088.493} C_VEL
LIN {X 0,Y 383.01,Z 255.778,A -85,B 0,C 180,E1 -12092.15,E2 -12092.15} C_VEL
LIN {X 0,Y 383.012,Z 255.773,A -85,B 0,C 180,E1 -12094.669,E2 -12094.669} C_VEL
LIN {X 0,Y 382.998,Z 255.78,A -85,B 0,C 180,E1 -12097.903,E2 -12097.903} C_VEL
LIN {X 0,Y 382.971,Z 255.78,A -85,B 0,C 180,E1 -12101.349,E2 -12101.349} C_VEL
LIN {X 0,Y 382.995,Z 255.776,A -85,B 0,C 180,E1 -12104.303,E2 -12104.303} C_VEL
LIN {X 0,Y 382.982,Z 255.779,A -85,B 0,C 180,E1 -12107.236,E2 -12107.236} C_VEL
LIN {X 0,Y 382.986,Z 255.775,A -85,B 0,C 180,E1 -12110.419,E2 -12110.419} C_VEL
LIN {X 0,Y 382.968,Z 255.784,A -85,B 0,C 180,E1 -12112.728,E2 -12112.728} C_VEL
LIN {X 0,Y 382.943,Z 255.923,A -85,B 0,C 180,E1 -12114.036,E2 -12114.036} C_VEL
LIN {X 0,Y 382.855,Z 258.808,A -85,B 0,C 180,E1 -12116.585,E2 -12116.585} C_VEL
LIN {X 0,Y 382.707,Z 262.435,A -85,B 0,C 180,E1 -12119.667,E2 -12119.667} C_VEL
LIN {X 0,Y 382.503,Z 266.028,A -85,B 0,C 180,E1 -12122.655,E2 -12122.655} C_VEL
LIN {X 0,Y 382.309,Z 270.407,A -85,B 0,C 180,E1 -12126.145,E2 -12126.145} C_VEL
LIN {X 0,Y 382.134,Z 275.047,A -85,B 0,C 180,E1 -12129.713,E2 -12129.713} C_VEL
LIN {X 0,Y 382.064,Z 277.058,A -85,B 0,C 180,E1 -12131.147,E2 -12131.147} C_VEL
LIN {X 0,Y 385.36,Z 290.339,A -85,B 0,C 180,E1 -12131.79,E2 -12131.79} C_VEL
LIN {X 0,Y 387.606,Z 301.523,A -85,B 0,C 180,E1 -12132.485,E2 -12132.485} C_VEL
LIN {X 0,Y 387.943,Z 305.903,A -85,B 0,C 180,E1 -12132.78,E2 -12132.78} C_VEL
LIN {X 0,Y 387.129,Z 317.785,A -85,B 0,C 180,E1 -12133.657,E2 -12133.657} C_VEL
LIN {X 0,Y 386.343,Z 328.555,A -85,B 0,C 180,E1 -12134.675,E2 -12134.675} C_VEL
LIN {X 0,Y 385.518,Z 337.793,A -85,B 0,C 180,E1 -12135.753,E2 -12135.753} C_VEL
LIN {X 0,Y 384.631,Z 346.973,A -85,B 0,C 180,E1 -12137.066,E2 -12137.066} C_VEL
LIN {X 0,Y 383.716,Z 355.888,A -85,B 0,C 180,E1 -12138.645,E2 -12138.645} C_VEL
LIN {X 0,Y 382.998,Z 363.063,A -85,B 0,C 180,E1 -12140.228,E2 -12140.228} C_VEL
LIN {X 0,Y 382.526,Z 367.901,A -85,B 0,C 180,E1 -12141.548,E2 -12141.548} C_VEL
LIN {X 0,Y 382.108,Z 373.095,A -85,B 0,C 180,E1 -12143.319,E2 -12143.319} C_VEL
LIN {X 0,Y 381.957,Z 376.197,A -85,B 0,C 180,E1 -12144.721,E2 -12144.721} C_VEL
LIN {X 0,Y 381.745,Z 378.059,A -85,B 0,C 180,E1 -12145.777,E2 -12145.777} C_VEL
LIN {X 0,Y 381.672,Z 379.458,A -85,B 0,C 180,E1 -12146.833,E2 -12146.833} C_VEL
LIN {X 0,Y 381.665,Z 380.452,A -85,B 0,C 180,E1 -12147.89,E2 -12147.89} C_VEL
LIN {X 0,Y 381.64,Z 381.297,A -85,B 0,C 180,E1 -12150,E2 -12150} C_VEL
LIN {X 0,Y 381.644,Z 381.108,A -85,B 0,C 180,E1 -12151.055,E2 -12151.055} C_VEL
LIN {X 0,Y 381.665,Z 380.524,A -85,B 0,C 180,E1 -12152.111,E2 -12152.111} C_VEL
LIN {X 0,Y 381.741,Z 378.204,A -85,B 0,C 180,E1 -12154.223,E2 -12154.223} C_VEL
LIN {X 0,Y 382.008,Z 375.336,A -85,B 0,C 180,E1 -12155.808,E2 -12155.808} C_VEL
LIN {X 0,Y 382.278,Z 371.451,A -85,B 0,C 180,E1 -12157.394,E2 -12157.394} C_VEL
LIN {X 0,Y 382.65,Z 366.439,A -85,B 0,C 180,E1 -12158.982,E2 -12158.982} C_VEL
LIN {X 0,Y 383.301,Z 360.125,A -85,B 0,C 180,E1 -12160.565,E2 -12160.565} C_VEL
LIN {X 0,Y 384.07,Z 352.221,A -85,B 0,C 180,E1 -12162.148,E2 -12162.148} C_VEL
LIN {X 0,Y 385.061,Z 342.387,A -85,B 0,C 180,E1 -12163.726,E2 -12163.726} C_VEL
LIN {X 0,Y 385.909,Z 333.171,A -85,B 0,C 180,E1 -12164.914,E2 -12164.914} C_VEL
LIN {X 0,Y 386.781,Z 321.843,A -85,B 0,C 180,E1 -12166.087,E2 -12166.087} C_VEL
LIN {X 0,Y 387.814,Z 309.741,A -85,B 0,C 180,E1 -12167.061,E2 -12167.061} C_VEL
LIN {X 0,Y 387.972,Z 303.712,A -85,B 0,C 180,E1 -12167.465,E2 -12167.465} C_VEL
LIN {X 0,Y 385.618,Z 291.588,A -85,B 0,C 180,E1 -12168.242,E2 -12168.242} C_VEL
LIN {X 0,Y 382.3,Z 278.366,A -85,B 0,C 180,E1 -12168.904,E2 -12168.904} C_VEL
LIN {X 0,Y 381.614,Z 277.124,A -85,B 0,C 180,E1 -12169.064,E2 -12169.064} C_VEL
LIN {X 0,Y 379.866,Z 276.266,A -85,B 0,C 180,E1 -12169.646,E2 -12169.646} C_VEL
LIN {X 0,Y 377.593,Z 275.045,A -85,B 0,C 180,E1 -12170.745,E2 -12170.745} C_VEL
LIN {X 0,Y 376.216,Z 274.244,A -85,B 0,C 180,E1 -12171.756,E2 -12171.756} C_VEL
LIN {X 0,Y 375.216,Z 271.826,A -85,B 0,C 180,E1 -12173.452,E2 -12173.452} C_VEL
LIN {X 0,Y 375.406,Z 267.793,A -85,B 0,C 180,E1 -12176.699,E2 -12176.699} C_VEL
LIN {X 0,Y 375.636,Z 263.44,A -85,B 0,C 180,E1 -12180.342,E2 -12180.342} C_VEL
LIN {X 0,Y 375.838,Z 259.084,A -85,B 0,C 180,E1 -12184.124,E2 -12184.124} C_VEL
LIN {X 0,Y 375.87,Z 256.668,A -85,B 0,C 180,E1 -12186.485,E2 -12186.485} C_VEL
LIN {X 0,Y 375.936,Z 256.654,A -85,B 0,C 180,E1 -12189.466,E2 -12189.466} C_VEL
LIN {X 0,Y 375.934,Z 256.655,A -85,B 0,C 180,E1 -12193.189,E2 -12193.189} C_VEL
LIN {X 0,Y 375.936,Z 256.656,A -85,B 0,C 180,E1 -12196.811,E2 -12196.811} C_VEL
LIN {X 0,Y 375.958,Z 256.654,A -85,B 0,C 180,E1 -12200.537,E2 -12200.537} C_VEL
LIN {X 0,Y 375.966,Z 256.651,A -85,B 0,C 180,E1 -12203.496,E2 -12203.496} C_VEL
LIN {X 0,Y 375.963,Z 256.655,A -85,B 0,C 180,E1 -12205.889,E2 -12205.889} C_VEL
LIN {X 0,Y 375.967,Z 256.654,A -85,B 0,C 180,E1 -12209.687,E2 -12209.687} C_VEL
LIN {X 0,Y 375.999,Z 256.649,A -85,B 0,C 180,E1 -12212.141,E2 -12212.141} C_VEL
LIN {X 0,Y 376.008,Z 256.645,A -85,B 0,C 180,E1 -12214.539,E2 -12214.539} C_VEL
LIN {X 0,Y 375.96,Z 256.652,A -85,B 0,C 180,E1 -12218.045,E2 -12218.045} C_VEL
LIN {X 0,Y 376.005,Z 256.651,A -85,B 0,C 180,E1 -12221.473,E2 -12221.473} C_VEL
LIN {X 0,Y 376.06,Z 256.64,A -85,B 0,C 180,E1 -12224.833,E2 -12224.833} C_VEL
LIN {X 0,Y 376.053,Z 256.639,A -85,B 0,C 180,E1 -12228.137,E2 -12228.137} C_VEL
LIN {X 0,Y 376.202,Z 256.621,A -85,B 0,C 180,E1 -12231.94,E2 -12231.94} C_VEL
LIN {X 0,Y 376.159,Z 256.628,A -85,B 0,C 180,E1 -12234.64,E2 -12234.64} C_VEL
LIN {X 0,Y 376.344,Z 256.603,A -85,B 0,C 180,E1 -12237.86,E2 -12237.86} C_VEL
LIN {X 0,Y 376.276,Z 256.615,A -85,B 0,C 180,E1 -12241.07,E2 -12241.07} C_VEL
LIN {X 0,Y 376.187,Z 256.624,A -85,B 0,C 180,E1 -12243.213,E2 -12243.213} C_VEL
LIN {X 0,Y 376.232,Z 256.622,A -85,B 0,C 180,E1 -12246.435,E2 -12246.435} C_VEL
LIN {X 0,Y 376.111,Z 256.632,A -85,B 0,C 180,E1 -12249.682,E2 -12249.682} C_VEL
LIN {X 0,Y 376.092,Z 256.635,A -85,B 0,C 180,E1 -12253.657,E2 -12253.657} C_VEL
LIN {X 0,Y 376.047,Z 256.641,A -85,B 0,C 180,E1 -12257.607,E2 -12257.607} C_VEL
LIN {X 0,Y 375.981,Z 256.649,A -85,B 0,C 180,E1 -12260.832,E2 -12260.832} C_VEL
LIN {X 0,Y 375.961,Z 256.653,A -85,B 0,C 180,E1 -12264.284,E2 -12264.284} C_VEL
LIN {X 0,Y 375.936,Z 256.659,A -85,B 0,C 180,E1 -12267.864,E2 -12267.864} C_VEL
LIN {X 0,Y 375.96,Z 256.656,A -85,B 0,C 180,E1 -12271.562,E2 -12271.562} C_VEL
LIN {X 0,Y 375.959,Z 256.656,A -85,B 0,C 180,E1 -12275.415,E2 -12275.415} C_VEL
LIN {X 0,Y 375.937,Z 256.654,A -85,B 0,C 180,E1 -12278.263,E2 -12278.263} C_VEL
LIN {X 0,Y 375.919,Z 256.66,A -85,B 0,C 180,E1 -12281.598,E2 -12281.598} C_VEL
LIN {X 0,Y 375.928,Z 256.66,A -85,B 0,C 180,E1 -12284.731,E2 -12284.731} C_VEL
LIN {X 0,Y 375.989,Z 256.726,A -85,B 0,C 180,E1 -12287.707,E2 -12287.707} C_VEL
LIN {X 0,Y 376.737,Z 261.002,A -85,B 0,C 180,E1 -12290.634,E2 -12290.634} C_VEL
LIN {X 0,Y 377.29,Z 265.289,A -85,B 0,C 180,E1 -12293.41,E2 -12293.41} C_VEL
LIN {X 0,Y 377.329,Z 267.938,A -85,B 0,C 180,E1 -12295.038,E2 -12295.038} C_VEL
LIN {X 0,Y 376.8,Z 273.883,A -85,B 0,C 180,E1 -12298.516,E2 -12298.516} C_VEL
LIN {X 0,Y 376.153,Z 280.347,A -85,B 0,C 180,E1 -12302.154,E2 -12302.154} C_VEL
LIN {X 0,Y 375.711,Z 286.753,A -85,B 0,C 180,E1 -12305.699,E2 -12305.699} C_VEL
LIN {X 0,Y 375.339,Z 293.107,A -85,B 0,C 180,E1 -12309.16,E2 -12309.16} C_VEL
LIN {X 0,Y 375.207,Z 296.122,A -85,B 0,C 180,E1 -12310.706,E2 -12310.706} C_VEL
LIN {X 0,Y 377.836,Z 309.351,A -85,B 0,C 180,E1 -12311.294,E2 -12311.294} C_VEL
LIN {X 0,Y 379.611,Z 321.391,A -85,B 0,C 180,E1 -12312.004,E2 -12312.004} C_VEL
LIN {X 0,Y 380.408,Z 331.217,A -85,B 0,C 180,E1 -12312.706,E2 -12312.706} C_VEL
LIN {X 0,Y 379.276,Z 343.506,A -85,B 0,C 180,E1 -12313.724,E2 -12313.724} C_VEL
LIN {X 0,Y 378.214,Z 354.751,A -85,B 0,C 180,E1 -12314.921,E2 -12314.921} C_VEL
LIN {X 0,Y 377.321,Z 364.718,A -85,B 0,C 180,E1 -12316.262,E2 -12316.262} C_VEL
LIN {X 0,Y 376.558,Z 372.893,A -85,B 0,C 180,E1 -12317.606,E2 -12317.606} C_VEL
LIN {X 0,Y 375.708,Z 380.913,A -85,B 0,C 180,E1 -12319.219,E2 -12319.219} C_VEL
LIN {X 0,Y 375.185,Z 387.348,A -85,B 0,C 180,E1 -12320.838,E2 -12320.838} C_VEL
LIN {X 0,Y 374.798,Z 392.459,A -85,B 0,C 180,E1 -12322.457,E2 -12322.457} C_VEL
LIN {X 0,Y 374.588,Z 396.103,A -85,B 0,C 180,E1 -12323.925,E2 -12323.925} C_VEL
LIN {X 0,Y 374.551,Z 399.365,A -85,B 0,C 180,E1 -12325.695,E2 -12325.695} C_VEL
LIN {X 0,Y 374.459,Z 401.756,A -85,B 0,C 180,E1 -12327.849,E2 -12327.849} C_VEL
LIN {X 0,Y 374.517,Z 402.366,A -85,B 0,C 180,E1 -12328.925,E2 -12328.925} C_VEL
LIN {X 0,Y 374.554,Z 402.582,A -85,B 0,C 180,E1 -12330,E2 -12330} C_VEL
LIN {X 0,Y 374.517,Z 402.363,A -85,B 0,C 180,E1 -12331.075,E2 -12331.075} C_VEL
LIN {X 0,Y 374.461,Z 400.753,A -85,B 0,C 180,E1 -12333.228,E2 -12333.228} C_VEL
LIN {X 0,Y 374.529,Z 399.354,A -85,B 0,C 180,E1 -12334.305,E2 -12334.305} C_VEL
LIN {X 0,Y 374.582,Z 396.104,A -85,B 0,C 180,E1 -12336.065,E2 -12336.065} C_VEL
LIN {X 0,Y 374.798,Z 392.432,A -85,B 0,C 180,E1 -12337.542,E2 -12337.542} C_VEL
LIN {X 0,Y 375.233,Z 386.314,A -85,B 0,C 180,E1 -12339.432,E2 -12339.432} C_VEL
LIN {X 0,Y 375.796,Z 379.632,A -85,B 0,C 180,E1 -12341.051,E2 -12341.051} C_VEL
LIN {X 0,Y 376.678,Z 371.346,A -85,B 0,C 180,E1 -12342.664,E2 -12342.664} C_VEL
LIN {X 0,Y 377.482,Z 362.85,A -85,B 0,C 180,E1 -12344.007,E2 -12344.007} C_VEL
LIN {X 0,Y 378.437,Z 352.353,A -85,B 0,C 180,E1 -12345.345,E2 -12345.345} C_VEL
LIN {X 0,Y 379.546,Z 340.542,A -85,B 0,C 180,E1 -12346.541,E2 -12346.541} C_VEL
LIN {X 0,Y 380.415,Z 329.795,A -85,B 0,C 180,E1 -12347.391,E2 -12347.391} C_VEL
LIN {X 0,Y 379.145,Z 317.906,A -85,B 0,C 180,E1 -12348.208,E2 -12348.208} C_VEL
LIN {X 0,Y 377.168,Z 305.962,A -85,B 0,C 180,E1 -12348.864,E2 -12348.864} C_VEL
LIN {X 0,Y 375.178,Z 295.91,A -85,B 0,C 180,E1 -12349.314,E2 -12349.314} C_VEL
LIN {X 0,Y 375.531,Z 289.93,A -85,B 0,C 180,E1 -12352.56,E2 -12352.56} C_VEL
LIN {X 0,Y 375.953,Z 283.279,A -85,B 0,C 180,E1 -12356.194,E2 -12356.194} C_VEL
LIN {X 0,Y 376.565,Z 275.988,A -85,B 0,C 180,E1 -12360.259,E2 -12360.259} C_VEL
LIN {X 0,Y 377.2,Z 269.54,A -85,B 0,C 180,E1 -12363.984,E2 -12363.984} C_VEL
LIN {X 0,Y 377.264,Z 265.244,A -85,B 0,C 180,E1 -12366.593,E2 -12366.593} C_VEL
LIN {X 0,Y 376.725,Z 260.963,A -85,B 0,C 180,E1 -12369.367,E2 -12369.367} C_VEL
LIN {X 0,Y 375.963,Z 256.66,A -85,B 0,C 180,E1 -12372.382,E2 -12372.382} C_VEL
LIN {X 0,Y 375.929,Z 256.658,A -85,B 0,C 180,E1 -12376.234,E2 -12376.234} C_VEL
LIN {X 0,Y 375.939,Z 256.654,A -85,B 0,C 180,E1 -12380.039,E2 -12380.039} C_VEL
LIN {X 0,Y 375.964,Z 256.65,A -85,B 0,C 180,E1 -12383.496,E2 -12383.496} C_VEL
LIN {X 0,Y 375.961,Z 256.652,A -85,B 0,C 180,E1 -12385.889,E2 -12385.889} C_VEL
LIN {X 0,Y 375.963,Z 256.652,A -85,B 0,C 180,E1 -12389.687,E2 -12389.687} C_VEL
LIN {X 0,Y 375.935,Z 256.659,A -85,B 0,C 180,E1 -12392.136,E2 -12392.136} C_VEL
LIN {X 0,Y 375.96,Z 256.653,A -85,B 0,C 180,E1 -12395.716,E2 -12395.716} C_VEL
LIN {X 0,Y 375.999,Z 256.646,A -85,B 0,C 180,E1 -12399.198,E2 -12399.198} C_VEL
LIN {X 0,Y 376.052,Z 256.64,A -85,B 0,C 180,E1 -12402.601,E2 -12402.601} C_VEL
LIN {X 0,Y 376.091,Z 256.635,A -85,B 0,C 180,E1 -12406.342,E2 -12406.342} C_VEL
LIN {X 0,Y 376.113,Z 256.632,A -85,B 0,C 180,E1 -12410.318,E2 -12410.318} C_VEL
LIN {X 0,Y 376.23,Z 256.622,A -85,B 0,C 180,E1 -12413.565,E2 -12413.565} C_VEL
LIN {X 0,Y 376.353,Z 256.603,A -85,B 0,C 180,E1 -12417.86,E2 -12417.86} C_VEL
LIN {X 0,Y 376.485,Z 256.586,A -85,B 0,C 180,E1 -12420,E2 -12420} C_VEL
LIN {X 0,Y 376.342,Z 256.603,A -85,B 0,C 180,E1 -12422.14,E2 -12422.14} C_VEL
LIN {X 0,Y 376.206,Z 256.62,A -85,B 0,C 180,E1 -12426.603,E2 -12426.603} C_VEL
LIN {X 0,Y 376.116,Z 256.632,A -85,B 0,C 180,E1 -12429.682,E2 -12429.682} C_VEL
LIN {X 0,Y 376.091,Z 256.635,A -85,B 0,C 180,E1 -12433.658,E2 -12433.658} C_VEL
LIN {X 0,Y 376.034,Z 256.642,A -85,B 0,C 180,E1 -12437.4,E2 -12437.4} C_VEL
LIN {X 0,Y 375.98,Z 256.651,A -85,B 0,C 180,E1 -12440.832,E2 -12440.832} C_VEL
LIN {X 0,Y 375.99,Z 256.652,A -85,B 0,C 180,E1 -12444.282,E2 -12444.282} C_VEL
LIN {X 0,Y 376.021,Z 256.646,A -85,B 0,C 180,E1 -12446.652,E2 -12446.652} C_VEL
LIN {X 0,Y 375.972,Z 256.65,A -85,B 0,C 180,E1 -12449.079,E2 -12449.079} C_VEL
LIN {X 0,Y 375.949,Z 256.653,A -85,B 0,C 180,E1 -12452.829,E2 -12452.829} C_VEL
LIN {X 0,Y 375.951,Z 256.653,A -85,B 0,C 180,E1 -12455.416,E2 -12455.416} C_VEL
LIN {X 0,Y 375.972,Z 256.652,A -85,B 0,C 180,E1 -12458.27,E2 -12458.27} C_VEL
LIN {X 0,Y 375.925,Z 256.659,A -85,B 0,C 180,E1 -12461.599,E2 -12461.599} C_VEL
LIN {X 0,Y 375.925,Z 256.655,A -85,B 0,C 180,E1 -12464.731,E2 -12464.731} C_VEL
LIN {X 0,Y 375.908,Z 256.663,A -85,B 0,C 180,E1 -12467.696,E2 -12467.696} C_VEL
LIN {X 0,Y 375.935,Z 256.654,A -85,B 0,C 180,E1 -12470.534,E2 -12470.534} C_VEL
LIN {X 0,Y 375.903,Z 256.663,A -85,B 0,C 180,E1 -12473.508,E2 -12473.508} C_VEL
LIN {X 0,Y 375.901,Z 258.38,A -85,B 0,C 180,E1 -12475.35,E2 -12475.35} C_VEL
LIN {X 0,Y 375.729,Z 261.854,A -85,B 0,C 180,E1 -12478.417,E2 -12478.417} C_VEL
LIN {X 0,Y 375.515,Z 266.194,A -85,B 0,C 180,E1 -12482.103,E2 -12482.103} C_VEL
LIN {X 0,Y 375.255,Z 270.583,A -85,B 0,C 180,E1 -12485.668,E2 -12485.668} C_VEL
LIN {X 0,Y 375.078,Z 275.021,A -85,B 0,C 180,E1 -12489.145,E2 -12489.145} C_VEL
LIN {X 0,Y 375.018,Z 277.173,A -85,B 0,C 180,E1 -12490.775,E2 -12490.775} C_VEL
LIN {X 0,Y 378.343,Z 290.613,A -85,B 0,C 180,E1 -12491.443,E2 -12491.443} C_VEL
LIN {X 0,Y 380.749,Z 302.304,A -85,B 0,C 180,E1 -12492.195,E2 -12492.195} C_VEL
LIN {X 0,Y 381.159,Z 306.397,A -85,B 0,C 180,E1 -12492.483,E2 -12492.483} C_VEL
LIN {X 0,Y 380.317,Z 317.991,A -85,B 0,C 180,E1 -12493.356,E2 -12493.356} C_VEL
LIN {X 0,Y 379.493,Z 328.544,A -85,B 0,C 180,E1 -12494.369,E2 -12494.369} C_VEL
LIN {X 0,Y 378.632,Z 337.997,A -85,B 0,C 180,E1 -12495.488,E2 -12495.488} C_VEL
LIN {X 0,Y 377.704,Z 347.176,A -85,B 0,C 180,E1 -12496.824,E2 -12496.824} C_VEL
LIN {X 0,Y 376.76,Z 356.09,A -85,B 0,C 180,E1 -12498.432,E2 -12498.432} C_VEL
LIN {X 0,Y 376.01,Z 363.264,A -85,B 0,C 180,E1 -12500.044,E2 -12500.044} C_VEL
LIN {X 0,Y 375.509,Z 368.103,A -85,B 0,C 180,E1 -12501.389,E2 -12501.389} C_VEL
LIN {X 0,Y 375.046,Z 373.56,A -85,B 0,C 180,E1 -12503.301,E2 -12503.301} C_VEL
LIN {X 0,Y 374.883,Z 376.398,A -85,B 0,C 180,E1 -12504.622,E2 -12504.622} C_VEL
LIN {X 0,Y 374.679,Z 378.259,A -85,B 0,C 180,E1 -12505.697,E2 -12505.697} C_VEL
LIN {X 0,Y 374.582,Z 379.658,A -85,B 0,C 180,E1 -12506.773,E2 -12506.773} C_VEL
LIN {X 0,Y 374.568,Z 380.652,A -85,B 0,C 180,E1 -12507.85,E2 -12507.85} C_VEL
LIN {X 0,Y 374.555,Z 381.497,A -85,B 0,C 180,E1 -12510,E2 -12510} C_VEL
LIN {X 0,Y 374.546,Z 381.308,A -85,B 0,C 180,E1 -12511.075,E2 -12511.075} C_VEL
LIN {X 0,Y 374.567,Z 380.724,A -85,B 0,C 180,E1 -12512.151,E2 -12512.151} C_VEL
LIN {X 0,Y 374.674,Z 378.402,A -85,B 0,C 180,E1 -12514.303,E2 -12514.303} C_VEL
LIN {X 0,Y 374.952,Z 375.535,A -85,B 0,C 180,E1 -12515.917,E2 -12515.917} C_VEL
LIN {X 0,Y 375.235,Z 371.65,A -85,B 0,C 180,E1 -12517.534,E2 -12517.534} C_VEL
LIN {X 0,Y 375.639,Z 366.637,A -85,B 0,C 180,E1 -12519.151,E2 -12519.151} C_VEL
LIN {X 0,Y 376.306,Z 360.323,A -85,B 0,C 180,E1 -12520.764,E2 -12520.764} C_VEL
LIN {X 0,Y 377.105,Z 352.419,A -85,B 0,C 180,E1 -12522.376,E2 -12522.376} C_VEL
LIN {X 0,Y 378.168,Z 342.584,A -85,B 0,C 180,E1 -12523.981,E2 -12523.981} C_VEL
LIN {X 0,Y 379.12,Z 332.853,A -85,B 0,C 180,E1 -12525.248,E2 -12525.248} C_VEL
LIN {X 0,Y 379.97,Z 322.038,A -85,B 0,C 180,E1 -12526.384,E2 -12526.384} C_VEL
LIN {X 0,Y 381.027,Z 310.063,A -85,B 0,C 180,E1 -12527.364,E2 -12527.364} C_VEL
LIN {X 0,Y 381.105,Z 304.38,A -85,B 0,C 180,E1 -12527.761,E2 -12527.761} C_VEL
LIN {X 0,Y 378.777,Z 292.383,A -85,B 0,C 180,E1 -12528.555,E2 -12528.555} C_VEL
LIN {X 0,Y 375.501,Z 279.314,A -85,B 0,C 180,E1 -12529.236,E2 -12529.236} C_VEL
LIN {X 0,Y 375.008,Z 277.134,A -85,B 0,C 180,E1 -12529.358,E2 -12529.358} C_VEL
LIN {X 0,Y 375.194,Z 272.188,A -85,B 0,C 180,E1 -12533.164,E2 -12533.164} C_VEL
LIN {X 0,Y 375.216,Z 271.826,A -85,B 0,C 180,E1 -12533.452,E2 -12533.452} C_VEL
LIN {X 0,Y 374.555,Z 270.805,A -85,B 0,C 180,E1 -12534.335,E2 -12534.335} C_VEL
LIN {X 0,Y 371.759,Z 269.342,A -85,B 0,C 180,E1 -12535.779,E2 -12535.779} C_VEL
LIN {X 0,Y 369.434,Z 268.198,A -85,B 0,C 180,E1 -12536.948,E2 -12536.948} C_VEL
LIN {X 0,Y 368.487,Z 267.236,A -85,B 0,C 180,E1 -12537.847,E2 -12537.847} C_VEL
LIN {X 0,Y 368.437,Z 266.882,A -85,B 0,C 180,E1 -12538.151,E2 -12538.151} C_VEL
LIN {X 0,Y 368.63,Z 263.602,A -85,B 0,C 180,E1 -12540.982,E2 -12540.982} C_VEL
LIN {X 0,Y 368.836,Z 259.104,A -85,B 0,C 180,E1 -12544.98,E2 -12544.98} C_VEL
LIN {X 0,Y 368.807,Z 257.77,A -85,B 0,C 180,E1 -12546.21,E2 -12546.21} C_VEL
LIN {X 0,Y 368.874,Z 257.536,A -85,B 0,C 180,E1 -12548.957,E2 -12548.957} C_VEL
LIN {X 0,Y 368.872,Z 257.535,A -85,B 0,C 180,E1 -12552.007,E2 -12552.007} C_VEL
LIN {X 0,Y 368.879,Z 257.533,A -85,B 0,C 180,E1 -12555.175,E2 -12555.175} C_VEL
LIN {X 0,Y 368.877,Z 257.538,A -85,B 0,C 180,E1 -12558.176,E2 -12558.176} C_VEL
LIN {X 0,Y 368.907,Z 257.529,A -85,B 0,C 180,E1 -12561.361,E2 -12561.361} C_VEL
LIN {X 0,Y 368.939,Z 257.525,A -85,B 0,C 180,E1 -12565.147,E2 -12565.147} C_VEL
LIN {X 0,Y 368.932,Z 257.526,A -85,B 0,C 180,E1 -12569.047,E2 -12569.047} C_VEL
LIN {X 0,Y 368.982,Z 257.524,A -85,B 0,C 180,E1 -12571.564,E2 -12571.564} C_VEL
LIN {X 0,Y 369.002,Z 257.52,A -85,B 0,C 180,E1 -12574.02,E2 -12574.02} C_VEL
LIN {X 0,Y 368.925,Z 257.533,A -85,B 0,C 180,E1 -12577.604,E2 -12577.604} C_VEL
LIN {X 0,Y 368.956,Z 257.526,A -85,B 0,C 180,E1 -12581.106,E2 -12581.106} C_VEL
LIN {X 0,Y 368.998,Z 257.518,A -85,B 0,C 180,E1 -12584.535,E2 -12584.535} C_VEL
LIN {X 0,Y 369.008,Z 257.517,A -85,B 0,C 180,E1 -12587.907,E2 -12587.907} C_VEL
LIN {X 0,Y 369.095,Z 257.511,A -85,B 0,C 180,E1 -12591.238,E2 -12591.238} C_VEL
LIN {X 0,Y 369.132,Z 257.503,A -85,B 0,C 180,E1 -12594.537,E2 -12594.537} C_VEL
LIN {X 0,Y 369.308,Z 257.479,A -85,B 0,C 180,E1 -12597.819,E2 -12597.819} C_VEL
LIN {X 0,Y 369.244,Z 257.49,A -85,B 0,C 180,E1 -12601.091,E2 -12601.091} C_VEL
LIN {X 0,Y 369.319,Z 257.479,A -85,B 0,C 180,E1 -12602.181,E2 -12602.181} C_VEL
LIN {X 0,Y 369.19,Z 257.5,A -85,B 0,C 180,E1 -12606.558,E2 -12606.558} C_VEL
LIN {X 0,Y 369.061,Z 257.511,A -85,B 0,C 180,E1 -12609.868,E2 -12609.868} C_VEL
LIN {X 0,Y 369.039,Z 257.514,A -85,B 0,C 180,E1 -12613.772,E2 -12613.772} C_VEL
LIN {X 0,Y 369.004,Z 257.519,A -85,B 0,C 180,E1 -12617.768,E2 -12617.768} C_VEL
LIN {X 0,Y 368.912,Z 257.529,A -85,B 0,C 180,E1 -12621.221,E2 -12621.221} C_VEL
LIN {X 0,Y 368.921,Z 257.533,A -85,B 0,C 180,E1 -12623.878,E2 -12623.878} C_VEL
LIN {X 0,Y 368.873,Z 257.534,A -85,B 0,C 180,E1 -12627.211,E2 -12627.211} C_VEL
LIN {X 0,Y 368.931,Z 257.527,A -85,B 0,C 180,E1 -12630.953,E2 -12630.953} C_VEL
LIN {X 0,Y 368.931,Z 257.527,A -85,B 0,C 180,E1 -12635.001,E2 -12635.001} C_VEL
LIN {X 0,Y 368.878,Z 257.533,A -85,B 0,C 180,E1 -12638.634,E2 -12638.634} C_VEL
LIN {X 0,Y 368.872,Z 257.534,A -85,B 0,C 180,E1 -12642.007,E2 -12642.007} C_VEL
LIN {X 0,Y 368.881,Z 257.538,A -85,B 0,C 180,E1 -12645.176,E2 -12645.176} C_VEL
LIN {X 0,Y 368.961,Z 257.583,A -85,B 0,C 180,E1 -12647.382,E2 -12647.382} C_VEL
LIN {X 0,Y 369.891,Z 263.011,A -85,B 0,C 180,E1 -12651.17,E2 -12651.17} C_VEL
LIN {X 0,Y 370.348,Z 267.295,A -85,B 0,C 180,E1 -12653.965,E2 -12653.965} C_VEL
LIN {X 0,Y 370.041,Z 271.767,A -85,B 0,C 180,E1 -12656.686,E2 -12656.686} C_VEL
LIN {X 0,Y 369.532,Z 276.959,A -85,B 0,C 180,E1 -12659.735,E2 -12659.735} C_VEL
LIN {X 0,Y 368.922,Z 283.641,A -85,B 0,C 180,E1 -12663.554,E2 -12663.554} C_VEL
LIN {X 0,Y 368.522,Z 289.77,A -85,B 0,C 180,E1 -12666.986,E2 -12666.986} C_VEL
LIN {X 0,Y 368.147,Z 295.93,A -85,B 0,C 180,E1 -12670.32,E2 -12670.32} C_VEL
LIN {X 0,Y 370.848,Z 309.152,A -85,B 0,C 180,E1 -12670.928,E2 -12670.928} C_VEL
LIN {X 0,Y 372.725,Z 321.884,A -85,B 0,C 180,E1 -12671.703,E2 -12671.703} C_VEL
LIN {X 0,Y 373.588,Z 331.085,A -85,B 0,C 180,E1 -12672.385,E2 -12672.385} C_VEL
LIN {X 0,Y 372.428,Z 343.309,A -85,B 0,C 180,E1 -12673.416,E2 -12673.416} C_VEL
LIN {X 0,Y 371.345,Z 354.554,A -85,B 0,C 180,E1 -12674.635,E2 -12674.635} C_VEL
LIN {X 0,Y 370.366,Z 364.518,A -85,B 0,C 180,E1 -12675.999,E2 -12675.999} C_VEL
LIN {X 0,Y 369.587,Z 372.694,A -85,B 0,C 180,E1 -12677.368,E2 -12677.368} C_VEL
LIN {X 0,Y 368.679,Z 380.713,A -85,B 0,C 180,E1 -12679.011,E2 -12679.011} C_VEL
LIN {X 0,Y 368.12,Z 387.148,A -85,B 0,C 180,E1 -12680.661,E2 -12680.661} C_VEL
LIN {X 0,Y 367.722,Z 392.259,A -85,B 0,C 180,E1 -12682.311,E2 -12682.311} C_VEL
LIN {X 0,Y 367.506,Z 396.2,A -85,B 0,C 180,E1 -12683.947,E2 -12683.947} C_VEL
LIN {X 0,Y 367.456,Z 399.165,A -85,B 0,C 180,E1 -12685.612,E2 -12685.612} C_VEL
LIN {X 0,Y 367.36,Z 401.557,A -85,B 0,C 180,E1 -12687.807,E2 -12687.807} C_VEL
LIN {X 0,Y 367.417,Z 402.166,A -85,B 0,C 180,E1 -12688.904,E2 -12688.904} C_VEL
LIN {X 0,Y 367.456,Z 402.382,A -85,B 0,C 180,E1 -12690,E2 -12690} C_VEL
LIN {X 0,Y 367.417,Z 402.163,A -85,B 0,C 180,E1 -12691.096,E2 -12691.096} C_VEL
LIN {X 0,Y 367.378,Z 400.553,A -85,B 0,C 180,E1 -12693.29,E2 -12693.29} C_VEL
LIN {X 0,Y 367.437,Z 399.154,A -85,B 0,C 180,E1 -12694.388,E2 -12694.388} C_VEL
LIN {X 0,Y 367.479,Z 396.259,A -85,B 0,C 180,E1 -12696.013,E2 -12696.013} C_VEL
LIN {X 0,Y 367.721,Z 392.23,A -85,B 0,C 180,E1 -12697.688,E2 -12697.688} C_VEL
LIN {X 0,Y 368.202,Z 386.112,A -85,B 0,C 180,E1 -12699.614,E2 -12699.614} C_VEL
LIN {X 0,Y 368.799,Z 379.429,A -85,B 0,C 180,E1 -12701.264,E2 -12701.264} C_VEL
LIN {X 0,Y 369.738,Z 371.144,A -85,B 0,C 180,E1 -12702.905,E2 -12702.905} C_VEL
LIN {X 0,Y 370.574,Z 362.647,A -85,B 0,C 180,E1 -12704.273,E2 -12704.273} C_VEL
LIN {X 0,Y 371.587,Z 352.15,A -85,B 0,C 180,E1 -12705.635,E2 -12705.635} C_VEL
LIN {X 0,Y 372.733,Z 340.338,A -85,B 0,C 180,E1 -12706.852,E2 -12706.852} C_VEL
LIN {X 0,Y 373.498,Z 329.723,A -85,B 0,C 180,E1 -12707.713,E2 -12707.713} C_VEL
LIN {X 0,Y 372.267,Z 318.481,A -85,B 0,C 180,E1 -12708.513,E2 -12708.513} C_VEL
LIN {X 0,Y 370.327,Z 306.464,A -85,B 0,C 180,E1 -12709.198,E2 -12709.198} C_VEL
LIN {X 0,Y 368.133,Z 295.707,A -85,B 0,C 180,E1 -12709.698,E2 -12709.698} C_VEL
LIN {X 0,Y 368.524,Z 289.744,A -85,B 0,C 180,E1 -12713.013,E2 -12713.013} C_VEL
LIN {X 0,Y 368.917,Z 283.605,A -85,B 0,C 180,E1 -12716.444,E2 -12716.444} C_VEL
LIN {X 0,Y 369.537,Z 276.917,A -85,B 0,C 180,E1 -12720.264,E2 -12720.264} C_VEL
LIN {X 0,Y 370.182,Z 270.451,A -85,B 0,C 180,E1 -12724.06,E2 -12724.06} C_VEL
LIN {X 0,Y 370.298,Z 267.247,A -85,B 0,C 180,E1 -12726.041,E2 -12726.041} C_VEL
LIN {X 0,Y 369.844,Z 262.962,A -85,B 0,C 180,E1 -12728.835,E2 -12728.835} C_VEL
LIN {X 0,Y 368.961,Z 257.531,A -85,B 0,C 180,E1 -12732.645,E2 -12732.645} C_VEL
LIN {X 0,Y 368.886,Z 257.538,A -85,B 0,C 180,E1 -12736.696,E2 -12736.696} C_VEL
LIN {X 0,Y 368.884,Z 257.532,A -85,B 0,C 180,E1 -12739.648,E2 -12739.648} C_VEL
LIN {X 0,Y 368.9,Z 257.531,A -85,B 0,C 180,E1 -12743.145,E2 -12743.145} C_VEL
LIN {X 0,Y 368.898,Z 257.536,A -85,B 0,C 180,E1 -12746.462,E2 -12746.462} C_VEL
LIN {X 0,Y 368.93,Z 257.527,A -85,B 0,C 180,E1 -12749.046,E2 -12749.046} C_VEL
LIN {X 0,Y 368.872,Z 257.534,A -85,B 0,C 180,E1 -12752.789,E2 -12752.789} C_VEL
LIN {X 0,Y 368.947,Z 257.527,A -85,B 0,C 180,E1 -12756.42,E2 -12756.42} C_VEL
LIN {X 0,Y 368.939,Z 257.531,A -85,B 0,C 180,E1 -12759.947,E2 -12759.947} C_VEL
LIN {X 0,Y 368.978,Z 257.523,A -85,B 0,C 180,E1 -12763.399,E2 -12763.399} C_VEL
LIN {X 0,Y 369.059,Z 257.51,A -85,B 0,C 180,E1 -12766.79,E2 -12766.79} C_VEL
LIN {X 0,Y 369.064,Z 257.511,A -85,B 0,C 180,E1 -12770.132,E2 -12770.132} C_VEL
LIN {X 0,Y 369.189,Z 257.5,A -85,B 0,C 180,E1 -12773.442,E2 -12773.442} C_VEL
LIN {X 0,Y 369.318,Z 257.48,A -85,B 0,C 180,E1 -12777.819,E2 -12777.819} C_VEL
LIN {X 0,Y 369.454,Z 257.461,A -85,B 0,C 180,E1 -12780,E2 -12780} C_VEL
LIN {X 0,Y 369.306,Z 257.479,A -85,B 0,C 180,E1 -12782.181,E2 -12782.181} C_VEL
LIN {X 0,Y 369.178,Z 257.497,A -85,B 0,C 180,E1 -12786.586,E2 -12786.586} C_VEL
LIN {X 0,Y 369.065,Z 257.509,A -85,B 0,C 180,E1 -12789.868,E2 -12789.868} C_VEL
LIN {X 0,Y 369.039,Z 257.513,A -85,B 0,C 180,E1 -12793.772,E2 -12793.772} C_VEL
LIN {X 0,Y 368.992,Z 257.519,A -85,B 0,C 180,E1 -12797.743,E2 -12797.743} C_VEL
LIN {X 0,Y 368.911,Z 257.529,A -85,B 0,C 180,E1 -12801.221,E2 -12801.221} C_VEL
LIN {X 0,Y 368.956,Z 257.526,A -85,B 0,C 180,E1 -12804.776,E2 -12804.776} C_VEL
LIN {X 0,Y 368.97,Z 257.521,A -85,B 0,C 180,E1 -12807.203,E2 -12807.203} C_VEL
LIN {X 0,Y 368.92,Z 257.529,A -85,B 0,C 180,E1 -12809.69,E2 -12809.69} C_VEL
LIN {X 0,Y 368.897,Z 257.53,A -85,B 0,C 180,E1 -12813.043,E2 -12813.043} C_VEL
LIN {X 0,Y 368.913,Z 257.533,A -85,B 0,C 180,E1 -12816.198,E2 -12816.198} C_VEL
LIN {X 0,Y 368.897,Z 257.53,A -85,B 0,C 180,E1 -12818.954,E2 -12818.954} C_VEL
LIN {X 0,Y 368.876,Z 257.537,A -85,B 0,C 180,E1 -12822.008,E2 -12822.008} C_VEL
LIN {X 0,Y 368.876,Z 257.535,A -85,B 0,C 180,E1 -12825.175,E2 -12825.175} C_VEL
LIN {X 0,Y 368.861,Z 257.536,A -85,B 0,C 180,E1 -12828.174,E2 -12828.174} C_VEL
LIN {X 0,Y 368.875,Z 257.538,A -85,B 0,C 180,E1 -12831.367,E2 -12831.367} C_VEL
LIN {X 0,Y 368.825,Z 257.648,A -85,B 0,C 180,E1 -12833.793,E2 -12833.793} C_VEL
LIN {X 0,Y 368.769,Z 260.576,A -85,B 0,C 180,E1 -12836.449,E2 -12836.449} C_VEL
LIN {X 0,Y 368.647,Z 263.538,A -85,B 0,C 180,E1 -12839.081,E2 -12839.081} C_VEL
LIN {X 0,Y 368.398,Z 267.827,A -85,B 0,C 180,E1 -12842.751,E2 -12842.751} C_VEL
LIN {X 0,Y 368.183,Z 272.256,A -85,B 0,C 180,E1 -12846.383,E2 -12846.383} C_VEL
LIN {X 0,Y 367.969,Z 277.367,A -85,B 0,C 180,E1 -12850.392,E2 -12850.392} C_VEL
LIN {X 0,Y 371.216,Z 290.207,A -85,B 0,C 180,E1 -12851.043,E2 -12851.043} C_VEL
LIN {X 0,Y 373.87,Z 303.04,A -85,B 0,C 180,E1 -12851.889,E2 -12851.889} C_VEL
LIN {X 0,Y 374.304,Z 308.086,A -85,B 0,C 180,E1 -12852.257,E2 -12852.257} C_VEL
LIN {X 0,Y 373.415,Z 319.766,A -85,B 0,C 180,E1 -12853.18,E2 -12853.18} C_VEL
LIN {X 0,Y 372.529,Z 330.609,A -85,B 0,C 180,E1 -12854.285,E2 -12854.285} C_VEL
LIN {X 0,Y 371.551,Z 340.158,A -85,B 0,C 180,E1 -12855.485,E2 -12855.485} C_VEL
LIN {X 0,Y 370.584,Z 349,A -85,B 0,C 180,E1 -12856.846,E2 -12856.846} C_VEL
LIN {X 0,Y 369.642,Z 357.623,A -85,B 0,C 180,E1 -12858.484,E2 -12858.484} C_VEL
LIN {X 0,Y 368.883,Z 364.497,A -85,B 0,C 180,E1 -12860.127,E2 -12860.127} C_VEL
LIN {X 0,Y 368.298,Z 369.999,A -85,B 0,C 180,E1 -12861.772,E2 -12861.772} C_VEL
LIN {X 0,Y 367.97,Z 374.315,A -85,B 0,C 180,E1 -12863.42,E2 -12863.42} C_VEL
LIN {X 0,Y 367.814,Z 376.599,A -85,B 0,C 180,E1 -12864.518,E2 -12864.518} C_VEL
LIN {X 0,Y 367.615,Z 378.459,A -85,B 0,C 180,E1 -12865.614,E2 -12865.614} C_VEL
LIN {X 0,Y 367.496,Z 379.859,A -85,B 0,C 180,E1 -12866.711,E2 -12866.711} C_VEL
LIN {X 0,Y 367.47,Z 380.852,A -85,B 0,C 180,E1 -12867.808,E2 -12867.808} C_VEL
LIN {X 0,Y 367.458,Z 381.696,A -85,B 0,C 180,E1 -12870,E2 -12870} C_VEL
LIN {X 0,Y 367.449,Z 381.507,A -85,B 0,C 180,E1 -12871.096,E2 -12871.096} C_VEL
LIN {X 0,Y 367.47,Z 380.923,A -85,B 0,C 180,E1 -12872.192,E2 -12872.192} C_VEL
LIN {X 0,Y 367.609,Z 378.601,A -85,B 0,C 180,E1 -12874.386,E2 -12874.386} C_VEL
LIN {X 0,Y 367.898,Z 375.734,A -85,B 0,C 180,E1 -12876.031,E2 -12876.031} C_VEL
LIN {X 0,Y 368.184,Z 371.849,A -85,B 0,C 180,E1 -12877.679,E2 -12877.679} C_VEL
LIN {X 0,Y 368.639,Z 366.835,A -85,B 0,C 180,E1 -12879.326,E2 -12879.326} C_VEL
LIN {X 0,Y 369.313,Z 360.521,A -85,B 0,C 180,E1 -12880.97,E2 -12880.97} C_VEL
LIN {X 0,Y 370.171,Z 352.616,A -85,B 0,C 180,E1 -12882.612,E2 -12882.612} C_VEL
LIN {X 0,Y 371.293,Z 342.78,A -85,B 0,C 180,E1 -12884.245,E2 -12884.245} C_VEL
LIN {X 0,Y 372.254,Z 333.049,A -85,B 0,C 180,E1 -12885.536,E2 -12885.536} C_VEL
LIN {X 0,Y 373.174,Z 322.232,A -85,B 0,C 180,E1 -12886.691,E2 -12886.691} C_VEL
LIN {X 0,Y 374.253,Z 310.37,A -85,B 0,C 180,E1 -12887.68,E2 -12887.68} C_VEL
LIN {X 0,Y 374.211,Z 304.977,A -85,B 0,C 180,E1 -12888.072,E2 -12888.072} C_VEL
LIN {X 0,Y 371.808,Z 292.94,A -85,B 0,C 180,E1 -12888.899,E2 -12888.899} C_VEL
LIN {X 0,Y 368.612,Z 280.008,A -85,B 0,C 180,E1 -12889.594,E2 -12889.594} C_VEL
LIN {X 0,Y 367.981,Z 277.318,A -85,B 0,C 180,E1 -12889.746,E2 -12889.746} C_VEL
LIN {X 0,Y 368.173,Z 272.37,A -85,B 0,C 180,E1 -12893.633,E2 -12893.633} C_VEL
LIN {X 0,Y 368.389,Z 267.96,A -85,B 0,C 180,E1 -12897.25,E2 -12897.25} C_VEL
LIN {X 0,Y 368.437,Z 266.882,A -85,B 0,C 180,E1 -12898.151,E2 -12898.151} C_VEL
LIN {X 0,Y 367.842,Z 265.907,A -85,B 0,C 180,E1 -12899.052,E2 -12899.052} C_VEL
LIN {X 0,Y 365.034,Z 264.569,A -85,B 0,C 180,E1 -12900.526,E2 -12900.526} C_VEL
LIN {X 0,Y 362.662,Z 263.538,A -85,B 0,C 180,E1 -12901.719,E2 -12901.719} C_VEL
LIN {X 0,Y 361.706,Z 262.651,A -85,B 0,C 180,E1 -12902.639,E2 -12902.639} C_VEL
LIN {X 0,Y 361.664,Z 262.313,A -85,B 0,C 180,E1 -12902.949,E2 -12902.949} C_VEL
LIN {X 0,Y 361.791,Z 259.364,A -85,B 0,C 180,E1 -12905.646,E2 -12905.646} C_VEL
LIN {X 0,Y 361.809,Z 258.418,A -85,B 0,C 180,E1 -12907.211,E2 -12907.211} C_VEL
LIN {X 0,Y 361.814,Z 258.416,A -85,B 0,C 180,E1 -12910.751,E2 -12910.751} C_VEL
LIN {X 0,Y 361.815,Z 258.418,A -85,B 0,C 180,E1 -12914.369,E2 -12914.369} C_VEL
LIN {X 0,Y 361.834,Z 258.411,A -85,B 0,C 180,E1 -12917.569,E2 -12917.569} C_VEL
LIN {X 0,Y 361.868,Z 258.406,A -85,B 0,C 180,E1 -12920.974,E2 -12920.974} C_VEL
LIN {X 0,Y 361.877,Z 258.406,A -85,B 0,C 180,E1 -12924.655,E2 -12924.655} C_VEL
LIN {X 0,Y 361.84,Z 258.411,A -85,B 0,C 180,E1 -12928.371,E2 -12928.371} C_VEL
LIN {X 0,Y 361.903,Z 258.402,A -85,B 0,C 180,E1 -12930.955,E2 -12930.955} C_VEL
LIN {X 0,Y 361.957,Z 258.398,A -85,B 0,C 180,E1 -12933.475,E2 -12933.475} C_VEL
LIN {X 0,Y 361.882,Z 258.406,A -85,B 0,C 180,E1 -12937.144,E2 -12937.144} C_VEL
LIN {X 0,Y 361.888,Z 258.404,A -85,B 0,C 180,E1 -12940.722,E2 -12940.722} C_VEL
LIN {X 0,Y 361.945,Z 258.396,A -85,B 0,C 180,E1 -12944.226,E2 -12944.226} C_VEL
LIN {X 0,Y 362.002,Z 258.39,A -85,B 0,C 180,E1 -12946.528,E2 -12946.528} C_VEL
LIN {X 0,Y 362.003,Z 258.389,A -85,B 0,C 180,E1 -12949.937,E2 -12949.937} C_VEL
LIN {X 0,Y 362.145,Z 258.375,A -85,B 0,C 180,E1 -12953.313,E2 -12953.313} C_VEL
LIN {X 0,Y 362.271,Z 258.356,A -85,B 0,C 180,E1 -12957.776,E2 -12957.776} C_VEL
LIN {X 0,Y 362.211,Z 258.366,A -85,B 0,C 180,E1 -12961.112,E2 -12961.112} C_VEL
LIN {X 0,Y 362.283,Z 258.356,A -85,B 0,C 180,E1 -12962.223,E2 -12962.223} C_VEL
LIN {X 0,Y 362.151,Z 258.376,A -85,B 0,C 180,E1 -12966.687,E2 -12966.687} C_VEL
LIN {X 0,Y 361.998,Z 258.392,A -85,B 0,C 180,E1 -12970.063,E2 -12970.063} C_VEL
LIN {X 0,Y 362,Z 258.391,A -85,B 0,C 180,E1 -12973.899,E2 -12973.899} C_VEL
LIN {X 0,Y 361.97,Z 258.397,A -85,B 0,C 180,E1 -12977.938,E2 -12977.938} C_VEL
LIN {X 0,Y 361.863,Z 258.409,A -85,B 0,C 180,E1 -12981.655,E2 -12981.655} C_VEL
LIN {X 0,Y 361.87,Z 258.406,A -85,B 0,C 180,E1 -12985.294,E2 -12985.294} C_VEL
LIN {X 0,Y 361.857,Z 258.408,A -85,B 0,C 180,E1 -12989.074,E2 -12989.074} C_VEL
LIN {X 0,Y 361.851,Z 258.409,A -85,B 0,C 180,E1 -12992.945,E2 -12992.945} C_VEL
LIN {X 0,Y 361.87,Z 258.411,A -85,B 0,C 180,E1 -12995.637,E2 -12995.637} C_VEL
LIN {X 0,Y 361.827,Z 258.413,A -85,B 0,C 180,E1 -12999.018,E2 -12999.018} C_VEL
LIN {X 0,Y 361.835,Z 258.412,A -85,B 0,C 180,E1 -13002.829,E2 -13002.829} C_VEL
LIN {X 0,Y 361.905,Z 258.49,A -85,B 0,C 180,E1 -13007.086,E2 -13007.086} C_VEL
LIN {X 0,Y 362.79,Z 263.683,A -85,B 0,C 180,E1 -13010.795,E2 -13010.795} C_VEL
LIN {X 0,Y 363.23,Z 267.155,A -85,B 0,C 180,E1 -13013.144,E2 -13013.144} C_VEL
LIN {X 0,Y 363.264,Z 270.374,A -85,B 0,C 180,E1 -13015.199,E2 -13015.199} C_VEL
LIN {X 0,Y 362.601,Z 276.832,A -85,B 0,C 180,E1 -13019.112,E2 -13019.112} C_VEL
LIN {X 0,Y 361.911,Z 283.955,A -85,B 0,C 180,E1 -13023.289,E2 -13023.289} C_VEL
LIN {X 0,Y 361.423,Z 290.64,A -85,B 0,C 180,E1 -13027.113,E2 -13027.113} C_VEL
LIN {X 0,Y 361.092,Z 295.545,A -85,B 0,C 180,E1 -13029.901,E2 -13029.901} C_VEL
LIN {X 0,Y 364.012,Z 309.879,A -85,B 0,C 180,E1 -13030.6,E2 -13030.6} C_VEL
LIN {X 0,Y 365.788,Z 321.685,A -85,B 0,C 180,E1 -13031.343,E2 -13031.343} C_VEL
LIN {X 0,Y 366.726,Z 332.106,A -85,B 0,C 180,E1 -13032.144,E2 -13032.144} C_VEL
LIN {X 0,Y 365.485,Z 344.534,A -85,B 0,C 180,E1 -13033.235,E2 -13033.235} C_VEL
LIN {X 0,Y 364.479,Z 354.356,A -85,B 0,C 180,E1 -13034.338,E2 -13034.338} C_VEL
LIN {X 0,Y 363.438,Z 364.32,A -85,B 0,C 180,E1 -13035.726,E2 -13035.726} C_VEL
LIN {X 0,Y 362.622,Z 372.495,A -85,B 0,C 180,E1 -13037.121,E2 -13037.121} C_VEL
LIN {X 0,Y 361.666,Z 380.514,A -85,B 0,C 180,E1 -13038.795,E2 -13038.795} C_VEL
LIN {X 0,Y 361.071,Z 386.948,A -85,B 0,C 180,E1 -13040.477,E2 -13040.477} C_VEL
LIN {X 0,Y 360.672,Z 392.059,A -85,B 0,C 180,E1 -13042.16,E2 -13042.16} C_VEL
LIN {X 0,Y 360.432,Z 396.246,A -85,B 0,C 180,E1 -13043.956,E2 -13043.956} C_VEL
LIN {X 0,Y 360.365,Z 398.966,A -85,B 0,C 180,E1 -13045.526,E2 -13045.526} C_VEL
LIN {X 0,Y 360.3,Z 400.361,A -85,B 0,C 180,E1 -13046.645,E2 -13046.645} C_VEL
LIN {X 0,Y 360.316,Z 401.967,A -85,B 0,C 180,E1 -13048.882,E2 -13048.882} C_VEL
LIN {X 0,Y 360.359,Z 402.183,A -85,B 0,C 180,E1 -13050,E2 -13050} C_VEL
LIN {X 0,Y 360.316,Z 401.962,A -85,B 0,C 180,E1 -13051.118,E2 -13051.118} C_VEL
LIN {X 0,Y 360.297,Z 400.353,A -85,B 0,C 180,E1 -13053.355,E2 -13053.355} C_VEL
LIN {X 0,Y 360.348,Z 398.953,A -85,B 0,C 180,E1 -13054.474,E2 -13054.474} C_VEL
LIN {X 0,Y 360.378,Z 396.385,A -85,B 0,C 180,E1 -13055.961,E2 -13055.961} C_VEL
LIN {X 0,Y 360.671,Z 392.029,A -85,B 0,C 180,E1 -13057.84,E2 -13057.84} C_VEL
LIN {X 0,Y 361.177,Z 385.91,A -85,B 0,C 180,E1 -13059.803,E2 -13059.803} C_VEL
LIN {X 0,Y 361.815,Z 379.227,A -85,B 0,C 180,E1 -13061.484,E2 -13061.484} C_VEL
LIN {X 0,Y 362.804,Z 370.942,A -85,B 0,C 180,E1 -13063.157,E2 -13063.157} C_VEL
LIN {X 0,Y 363.82,Z 361.168,A -85,B 0,C 180,E1 -13064.731,E2 -13064.731} C_VEL
LIN {X 0,Y 364.85,Z 350.769,A -85,B 0,C 180,E1 -13066.075,E2 -13066.075} C_VEL
LIN {X 0,Y 365.905,Z 340.133,A -85,B 0,C 180,E1 -13067.176,E2 -13067.176} C_VEL
LIN {X 0,Y 366.673,Z 330.816,A -85,B 0,C 180,E1 -13067.951,E2 -13067.951} C_VEL
LIN {X 0,Y 365.572,Z 320.206,A -85,B 0,C 180,E1 -13068.749,E2 -13068.749} C_VEL
LIN {X 0,Y 363.621,Z 307.858,A -85,B 0,C 180,E1 -13069.502,E2 -13069.502} C_VEL
LIN {X 0,Y 361.092,Z 295.522,A -85,B 0,C 180,E1 -13070.099,E2 -13070.099} C_VEL
LIN {X 0,Y 361.425,Z 290.615,A -85,B 0,C 180,E1 -13072.886,E2 -13072.886} C_VEL
LIN {X 0,Y 361.906,Z 283.93,A -85,B 0,C 180,E1 -13076.71,E2 -13076.71} C_VEL
LIN {X 0,Y 362.6,Z 276.794,A -85,B 0,C 180,E1 -13080.887,E2 -13080.887} C_VEL
LIN {X 0,Y 363.244,Z 270.317,A -85,B 0,C 180,E1 -13084.803,E2 -13084.803} C_VEL
LIN {X 0,Y 363.134,Z 266.157,A -85,B 0,C 180,E1 -13087.486,E2 -13087.486} C_VEL
LIN {X 0,Y 362.374,Z 261.286,A -85,B 0,C 180,E1 -13090.854,E2 -13090.854} C_VEL
LIN {X 0,Y 361.873,Z 258.412,A -85,B 0,C 180,E1 -13093.013,E2 -13093.013} C_VEL
LIN {X 0,Y 361.834,Z 258.412,A -85,B 0,C 180,E1 -13097.171,E2 -13097.171} C_VEL
LIN {X 0,Y 361.826,Z 258.413,A -85,B 0,C 180,E1 -13100.982,E2 -13100.982} C_VEL
LIN {X 0,Y 361.875,Z 258.409,A -85,B 0,C 180,E1 -13104.655,E2 -13104.655} C_VEL
LIN {X 0,Y 361.839,Z 258.415,A -85,B 0,C 180,E1 -13108.371,E2 -13108.371} C_VEL
LIN {X 0,Y 361.866,Z 258.407,A -85,B 0,C 180,E1 -13110.952,E2 -13110.952} C_VEL
LIN {X 0,Y 361.868,Z 258.407,A -85,B 0,C 180,E1 -13114.705,E2 -13114.705} C_VEL
LIN {X 0,Y 361.855,Z 258.41,A -85,B 0,C 180,E1 -13118.345,E2 -13118.345} C_VEL
LIN {X 0,Y 361.969,Z 258.397,A -85,B 0,C 180,E1 -13122.061,E2 -13122.061} C_VEL
LIN {X 0,Y 361.999,Z 258.392,A -85,B 0,C 180,E1 -13126.101,E2 -13126.101} C_VEL
LIN {X 0,Y 362,Z 258.392,A -85,B 0,C 180,E1 -13129.937,E2 -13129.937} C_VEL
LIN {X 0,Y 362.15,Z 258.375,A -85,B 0,C 180,E1 -13133.313,E2 -13133.313} C_VEL
LIN {X 0,Y 362.282,Z 258.356,A -85,B 0,C 180,E1 -13137.776,E2 -13137.776} C_VEL
LIN {X 0,Y 362.403,Z 258.34,A -85,B 0,C 180,E1 -13140,E2 -13140} C_VEL
LIN {X 0,Y 362.269,Z 258.356,A -85,B 0,C 180,E1 -13142.224,E2 -13142.224} C_VEL
LIN {X 0,Y 362.143,Z 258.374,A -85,B 0,C 180,E1 -13146.687,E2 -13146.687} C_VEL
LIN {X 0,Y 362.002,Z 258.389,A -85,B 0,C 180,E1 -13150.063,E2 -13150.063} C_VEL
LIN {X 0,Y 362,Z 258.39,A -85,B 0,C 180,E1 -13153.899,E2 -13153.899} C_VEL
LIN {X 0,Y 361.93,Z 258.402,A -85,B 0,C 180,E1 -13156.934,E2 -13156.934} C_VEL
LIN {X 0,Y 361.888,Z 258.409,A -85,B 0,C 180,E1 -13160.461,E2 -13160.461} C_VEL
LIN {X 0,Y 361.894,Z 258.406,A -85,B 0,C 180,E1 -13164.113,E2 -13164.113} C_VEL
LIN {X 0,Y 361.944,Z 258.399,A -85,B 0,C 180,E1 -13166.722,E2 -13166.722} C_VEL
LIN {X 0,Y 361.876,Z 258.41,A -85,B 0,C 180,E1 -13170.328,E2 -13170.328} C_VEL
LIN {X 0,Y 361.852,Z 258.412,A -85,B 0,C 180,E1 -13174.281,E2 -13174.281} C_VEL
LIN {X 0,Y 361.862,Z 258.407,A -85,B 0,C 180,E1 -13177.222,E2 -13177.222} C_VEL
LIN {X 0,Y 361.831,Z 258.41,A -85,B 0,C 180,E1 -13180.754,E2 -13180.754} C_VEL
LIN {X 0,Y 361.816,Z 258.413,A -85,B 0,C 180,E1 -13184.369,E2 -13184.369} C_VEL
LIN {X 0,Y 361.823,Z 258.417,A -85,B 0,C 180,E1 -13187.571,E2 -13187.571} C_VEL
LIN {X 0,Y 361.837,Z 258.415,A -85,B 0,C 180,E1 -13191.571,E2 -13191.571} C_VEL
LIN {X 0,Y 361.83,Z 258.417,A -85,B 0,C 180,E1 -13192.978,E2 -13192.978} C_VEL
LIN {X 0,Y 361.817,Z 259.587,A -85,B 0,C 180,E1 -13194.668,E2 -13194.668} C_VEL
LIN {X 0,Y 361.721,Z 262.169,A -85,B 0,C 180,E1 -13197.042,E2 -13197.042} C_VEL
LIN {X 0,Y 361.559,Z 265.084,A -85,B 0,C 180,E1 -13199.643,E2 -13199.643} C_VEL
LIN {X 0,Y 361.302,Z 269.541,A -85,B 0,C 180,E1 -13203.481,E2 -13203.481} C_VEL
LIN {X 0,Y 361.039,Z 273.897,A -85,B 0,C 180,E1 -13207.088,E2 -13207.088} C_VEL
LIN {X 0,Y 360.921,Z 277.598,A -85,B 0,C 180,E1 -13209.993,E2 -13209.993} C_VEL
LIN {X 0,Y 364.231,Z 290.526,A -85,B 0,C 180,E1 -13210.67,E2 -13210.67} C_VEL
LIN {X 0,Y 366.864,Z 303.011,A -85,B 0,C 180,E1 -13211.515,E2 -13211.515} C_VEL
LIN {X 0,Y 367.552,Z 308.469,A -85,B 0,C 180,E1 -13211.933,E2 -13211.933} C_VEL
LIN {X 0,Y 366.632,Z 319.971,A -85,B 0,C 180,E1 -13212.859,E2 -13212.859} C_VEL
LIN {X 0,Y 365.642,Z 331.422,A -85,B 0,C 180,E1 -13214.056,E2 -13214.056} C_VEL
LIN {X 0,Y 364.469,Z 342.305,A -85,B 0,C 180,E1 -13215.483,E2 -13215.483} C_VEL
LIN {X 0,Y 363.499,Z 350.8,A -85,B 0,C 180,E1 -13216.869,E2 -13216.869} C_VEL
LIN {X 0,Y 362.523,Z 359.053,A -85,B 0,C 180,E1 -13218.539,E2 -13218.539} C_VEL
LIN {X 0,Y 361.779,Z 365.7,A -85,B 0,C 180,E1 -13220.213,E2 -13220.213} C_VEL
LIN {X 0,Y 361.125,Z 371.788,A -85,B 0,C 180,E1 -13222.17,E2 -13222.17} C_VEL
LIN {X 0,Y 360.845,Z 375.427,A -85,B 0,C 180,E1 -13223.704,E2 -13223.704} C_VEL
LIN {X 0,Y 360.553,Z 378.659,A -85,B 0,C 180,E1 -13225.528,E2 -13225.528} C_VEL
LIN {X 0,Y 360.413,Z 380.059,A -85,B 0,C 180,E1 -13226.646,E2 -13226.646} C_VEL
LIN {X 0,Y 360.353,Z 381.664,A -85,B 0,C 180,E1 -13228.883,E2 -13228.883} C_VEL
LIN {X 0,Y 360.361,Z 381.896,A -85,B 0,C 180,E1 -13230,E2 -13230} C_VEL
LIN {X 0,Y 360.353,Z 381.707,A -85,B 0,C 180,E1 -13231.118,E2 -13231.118} C_VEL
LIN {X 0,Y 360.411,Z 380.157,A -85,B 0,C 180,E1 -13233.354,E2 -13233.354} C_VEL
LIN {X 0,Y 360.546,Z 378.8,A -85,B 0,C 180,E1 -13234.472,E2 -13234.472} C_VEL
LIN {X 0,Y 360.839,Z 375.665,A -85,B 0,C 180,E1 -13236.287,E2 -13236.287} C_VEL
LIN {X 0,Y 361.137,Z 372.048,A -85,B 0,C 180,E1 -13237.83,E2 -13237.83} C_VEL
LIN {X 0,Y 361.62,Z 367.034,A -85,B 0,C 180,E1 -13239.509,E2 -13239.509} C_VEL
LIN {X 0,Y 362.335,Z 360.719,A -85,B 0,C 180,E1 -13241.184,E2 -13241.184} C_VEL
LIN {X 0,Y 363.254,Z 352.813,A -85,B 0,C 180,E1 -13242.856,E2 -13242.856} C_VEL
LIN {X 0,Y 364.431,Z 342.976,A -85,B 0,C 180,E1 -13244.519,E2 -13244.519} C_VEL
LIN {X 0,Y 365.402,Z 333.435,A -85,B 0,C 180,E1 -13245.812,E2 -13245.812} C_VEL
LIN {X 0,Y 366.381,Z 322.427,A -85,B 0,C 180,E1 -13247.01,E2 -13247.01} C_VEL
LIN {X 0,Y 367.488,Z 310.68,A -85,B 0,C 180,E1 -13248.007,E2 -13248.007} C_VEL
LIN {X 0,Y 367.535,Z 306.862,A -85,B 0,C 180,E1 -13248.288,E2 -13248.288} C_VEL
LIN {X 0,Y 365.163,Z 294.721,A -85,B 0,C 180,E1 -13249.177,E2 -13249.177} C_VEL
LIN {X 0,Y 362.173,Z 282.319,A -85,B 0,C 180,E1 -13249.888,E2 -13249.888} C_VEL
LIN {X 0,Y 360.934,Z 277.52,A -85,B 0,C 180,E1 -13250.144,E2 -13250.144} C_VEL
LIN {X 0,Y 361.138,Z 272.559,A -85,B 0,C 180,E1 -13254.122,E2 -13254.122} C_VEL
LIN {X 0,Y 361.374,Z 268.134,A -85,B 0,C 180,E1 -13257.824,E2 -13257.824} C_VEL
LIN {X 0,Y 361.589,Z 264.236,A -85,B 0,C 180,E1 -13261.217,E2 -13261.217} C_VEL
LIN {X 0,Y 361.664,Z 262.313,A -85,B 0,C 180,E1 -13262.949,E2 -13262.949} C_VEL
LIN {X 0,Y 361.095,Z 261.385,A -85,B 0,C 180,E1 -13263.868,E2 -13263.868} C_VEL
LIN {X 0,Y 358.294,Z 260.146,A -85,B 0,C 180,E1 -13265.371,E2 -13265.371} C_VEL
LIN {X 0,Y 355.877,Z 259.526,A -85,B 0,C 180,E1 -13266.593,E2 -13266.593} C_VEL
LIN {X 0,Y 354.849,Z 259.309,A -85,B 0,C 180,E1 -13267.54,E2 -13267.54} C_VEL
LIN {X 0,Y 354.774,Z 259.292,A -85,B 0,C 180,E1 -13267.861,E2 -13267.861} C_VEL
LIN {X 0,Y 354.772,Z 259.29,A -85,B 0,C 180,E1 -13271.168,E2 -13271.168} C_VEL
LIN {X 0,Y 354.762,Z 259.296,A -85,B 0,C 180,E1 -13274.506,E2 -13274.506} C_VEL
LIN {X 0,Y 354.793,Z 259.288,A -85,B 0,C 180,E1 -13277.662,E2 -13277.662} C_VEL
LIN {X 0,Y 354.818,Z 259.286,A -85,B 0,C 180,E1 -13280.666,E2 -13280.666} C_VEL
LIN {X 0,Y 354.824,Z 259.287,A -85,B 0,C 180,E1 -13284.301,E2 -13284.301} C_VEL
LIN {X 0,Y 354.789,Z 259.291,A -85,B 0,C 180,E1 -13287.667,E2 -13287.667} C_VEL
LIN {X 0,Y 354.871,Z 259.278,A -85,B 0,C 180,E1 -13290.621,E2 -13290.621} C_VEL
LIN {X 0,Y 354.901,Z 259.276,A -85,B 0,C 180,E1 -13294.173,E2 -13294.173} C_VEL
LIN {X 0,Y 354.818,Z 259.287,A -85,B 0,C 180,E1 -13297.893,E2 -13297.893} C_VEL
LIN {X 0,Y 354.892,Z 259.277,A -85,B 0,C 180,E1 -13301.908,E2 -13301.908} C_VEL
LIN {X 0,Y 354.946,Z 259.269,A -85,B 0,C 180,E1 -13305.981,E2 -13305.981} C_VEL
LIN {X 0,Y 354.959,Z 259.268,A -85,B 0,C 180,E1 -13309.735,E2 -13309.735} C_VEL
LIN {X 0,Y 355.109,Z 259.253,A -85,B 0,C 180,E1 -13313.18,E2 -13313.18} C_VEL
LIN {X 0,Y 355.233,Z 259.233,A -85,B 0,C 180,E1 -13317.732,E2 -13317.732} C_VEL
LIN {X 0,Y 355.18,Z 259.242,A -85,B 0,C 180,E1 -13321.134,E2 -13321.134} C_VEL
LIN {X 0,Y 355.246,Z 259.233,A -85,B 0,C 180,E1 -13322.268,E2 -13322.268} C_VEL
LIN {X 0,Y 355.114,Z 259.251,A -85,B 0,C 180,E1 -13326.82,E2 -13326.82} C_VEL
LIN {X 0,Y 354.954,Z 259.271,A -85,B 0,C 180,E1 -13330.265,E2 -13330.265} C_VEL
LIN {X 0,Y 354.945,Z 259.271,A -85,B 0,C 180,E1 -13334.019,E2 -13334.019} C_VEL
LIN {X 0,Y 354.926,Z 259.276,A -85,B 0,C 180,E1 -13338.109,E2 -13338.109} C_VEL
LIN {X 0,Y 354.816,Z 259.29,A -85,B 0,C 180,E1 -13342.107,E2 -13342.107} C_VEL
LIN {X 0,Y 354.81,Z 259.291,A -85,B 0,C 180,E1 -13345.834,E2 -13345.834} C_VEL
LIN {X 0,Y 354.801,Z 259.291,A -85,B 0,C 180,E1 -13349.683,E2 -13349.683} C_VEL
LIN {X 0,Y 354.833,Z 259.288,A -85,B 0,C 180,E1 -13353.682,E2 -13353.682} C_VEL
LIN {X 0,Y 354.797,Z 259.287,A -85,B 0,C 180,E1 -13356.46,E2 -13356.46} C_VEL
LIN {X 0,Y 354.769,Z 259.296,A -85,B 0,C 180,E1 -13359.412,E2 -13359.412} C_VEL
LIN {X 0,Y 354.787,Z 259.29,A -85,B 0,C 180,E1 -13362.867,E2 -13362.867} C_VEL
LIN {X 0,Y 354.863,Z 259.48,A -85,B 0,C 180,E1 -13366.839,E2 -13366.839} C_VEL
LIN {X 0,Y 355.7,Z 264.335,A -85,B 0,C 180,E1 -13370.405,E2 -13370.405} C_VEL
LIN {X 0,Y 356.216,Z 268.097,A -85,B 0,C 180,E1 -13373.004,E2 -13373.004} C_VEL
LIN {X 0,Y 356.248,Z 271.294,A -85,B 0,C 180,E1 -13375.102,E2 -13375.102} C_VEL
LIN {X 0,Y 355.575,Z 277.71,A -85,B 0,C 180,E1 -13379.076,E2 -13379.076} C_VEL
LIN {X 0,Y 354.887,Z 284.292,A -85,B 0,C 180,E1 -13383.019,E2 -13383.019} C_VEL
LIN {X 0,Y 354.411,Z 290.452,A -85,B 0,C 180,E1 -13386.634,E2 -13386.634} C_VEL
LIN {X 0,Y 354.09,Z 295.335,A -85,B 0,C 180,E1 -13389.486,E2 -13389.486} C_VEL
LIN {X 0,Y 357.033,Z 309.75,A -85,B 0,C 180,E1 -13390.208,E2 -13390.208} C_VEL
LIN {X 0,Y 358.938,Z 322.16,A -85,B 0,C 180,E1 -13391.018,E2 -13391.018} C_VEL
LIN {X 0,Y 359.897,Z 331.909,A -85,B 0,C 180,E1 -13391.793,E2 -13391.793} C_VEL
